LIN {X 0,Y 202.976,Z 342.677,A -85,B 0,C 180,E1 -21997.686,E2 -21997.686} C_VEL
LIN {X 0,Y 206.775,Z 348.376,A -85,B 0,C 180,E1 -21999.696,E2 -21999.696} C_VEL
LIN {X 0,Y 211.34,Z 355.755,A -85,B 0,C 180,E1 -22001.921,E2 -22001.921} C_VEL
LIN {X 0,Y 216.534,Z 364.56,A -85,B 0,C 180,E1 -22004.233,E2 -22004.233} C_VEL
LIN {X 0,Y 221.924,Z 374.855,A -85,B 0,C 180,E1 -22006.449,E2 -22006.449} C_VEL
LIN {X 0,Y 227.529,Z 386.979,A -85,B 0,C 180,E1 -22008.613,E2 -22008.613} C_VEL
LIN {X 0,Y 230.022,Z 393.221,A -85,B 0,C 180,E1 -22009.55,E2 -22009.55} C_VEL
LIN {X 0,Y 230.632,Z 398.833,A -85,B 0,C 180,E1 -22009.954,E2 -22009.954} C_VEL
LIN {X 0,Y 229.742,Z 414.651,A -85,B 0,C 180,E1 -22010.427,E2 -22010.427} C_VEL
LIN {X 0,Y 228.926,Z 420.5,A -85,B 0,C 180,E1 -22010.473,E2 -22010.473} C_VEL
LIN {X 0,Y 223.579,Z 439.513,A -85,B 0,C 180,E1 -22010.007,E2 -22010.007} C_VEL
LIN {X 0,Y 222.491,Z 445.308,A -85,B 0,C 180,E1 -22010.121,E2 -22010.121} C_VEL
LIN {X 0,Y 220.529,Z 457.934,A -85,B 0,C 180,E1 -22010.845,E2 -22010.845} C_VEL
LIN {X 0,Y 217.724,Z 470.431,A -85,B 0,C 180,E1 -22011.877,E2 -22011.877} C_VEL
LIN {X 0,Y 214.297,Z 482.437,A -85,B 0,C 180,E1 -22013.235,E2 -22013.235} C_VEL
LIN {X 0,Y 210.551,Z 493.18,A -85,B 0,C 180,E1 -22014.844,E2 -22014.844} C_VEL
LIN {X 0,Y 206.238,Z 503.921,A -85,B 0,C 180,E1 -22016.958,E2 -22016.958} C_VEL
LIN {X 0,Y 202.158,Z 512.677,A -85,B 0,C 180,E1 -22019.149,E2 -22019.149} C_VEL
LIN {X 0,Y 197.802,Z 521.235,A -85,B 0,C 180,E1 -22021.914,E2 -22021.914} C_VEL
LIN {X 0,Y 193.915,Z 528.409,A -85,B 0,C 180,E1 -22024.968,E2 -22024.968} C_VEL
LIN {X 0,Y 190.389,Z 534.447,A -85,B 0,C 180,E1 -22028.336,E2 -22028.336} C_VEL
LIN {X 0,Y 187.771,Z 538.634,A -85,B 0,C 180,E1 -22031.448,E2 -22031.448} C_VEL
LIN {X 0,Y 185.687,Z 541.79,A -85,B 0,C 180,E1 -22034.635,E2 -22034.635} C_VEL
LIN {X 0,Y 184.75,Z 543.382,A -85,B 0,C 180,E1 -22036.805,E2 -22036.805} C_VEL
LIN {X 0,Y 184.038,Z 544.562,A -85,B 0,C 180,E1 -22038.991,E2 -22038.991} C_VEL
LIN {X 0,Y 183.222,Z 545.704,A -85,B 0,C 180,E1 -22043.391,E2 -22043.391} C_VEL
LIN {X 0,Y 183.133,Z 545.653,A -85,B 0,C 180,E1 -22046.191,E2 -22046.191} C_VEL
LIN {X 0,Y 183.342,Z 544.51,A -85,B 0,C 180,E1 -22049.998,E2 -22049.998} C_VEL
LIN {X 0,Y 183.16,Z 541.988,A -85,B 0,C 180,E1 -22053.935,E2 -22053.935} C_VEL
LIN {X 0,Y 183.374,Z 538.253,A -85,B 0,C 180,E1 -22057.707,E2 -22057.707} C_VEL
LIN {X 0,Y 183.903,Z 533.789,A -85,B 0,C 180,E1 -22061.014,E2 -22061.014} C_VEL
LIN {X 0,Y 184.844,Z 528.091,A -85,B 0,C 180,E1 -22064.306,E2 -22064.306} C_VEL
LIN {X 0,Y 186.496,Z 520.949,A -85,B 0,C 180,E1 -22067.544,E2 -22067.544} C_VEL
LIN {X 0,Y 188.388,Z 512.541,A -85,B 0,C 180,E1 -22070.564,E2 -22070.564} C_VEL
LIN {X 0,Y 189.713,Z 506.711,A -85,B 0,C 180,E1 -22072.314,E2 -22072.314} C_VEL
LIN {X 0,Y 191.746,Z 497.383,A -85,B 0,C 180,E1 -22074.638,E2 -22074.638} C_VEL
LIN {X 0,Y 193.876,Z 487.221,A -85,B 0,C 180,E1 -22076.651,E2 -22076.651} C_VEL
LIN {X 0,Y 196.128,Z 476.194,A -85,B 0,C 180,E1 -22078.344,E2 -22078.344} C_VEL
LIN {X 0,Y 197.847,Z 465.063,A -85,B 0,C 180,E1 -22079.674,E2 -22079.674} C_VEL
LIN {X 0,Y 199.457,Z 452.039,A -85,B 0,C 180,E1 -22080.796,E2 -22080.796} C_VEL
LIN {X 0,Y 200.468,Z 439.102,A -85,B 0,C 180,E1 -22081.503,E2 -22081.503} C_VEL
LIN {X 0,Y 202.387,Z 390.412,A -85,B 0,C 180,E1 -22083.182,E2 -22083.182} C_VEL
LIN {X 0,Y 199.567,Z 364.019,A -85,B 0,C 180,E1 -22084.672,E2 -22084.672} C_VEL
LIN {X 0,Y 193.84,Z 348.784,A -85,B 0,C 180,E1 -22086.254,E2 -22086.254} C_VEL
LIN {X 0,Y 188.083,Z 335.728,A -85,B 0,C 180,E1 -22087.863,E2 -22087.863} C_VEL
LIN {X 0,Y 186.801,Z 332.704,A -85,B 0,C 180,E1 -22088.273,E2 -22088.273} C_VEL
LIN {X 0,Y 185.491,Z 327.376,A -85,B 0,C 180,E1 -22091.228,E2 -22091.228} C_VEL
LIN {X 0,Y 185.456,Z 327.385,A -85,B 0,C 180,E1 -22096.053,E2 -22096.053} C_VEL
LIN {X 0,Y 185.484,Z 327.371,A -85,B 0,C 180,E1 -22099.9,E2 -22099.9} C_VEL
LIN {X 0,Y 185.539,Z 327.374,A -85,B 0,C 180,E1 -22102.695,E2 -22102.695} C_VEL
LIN {X 0,Y 185.54,Z 327.368,A -85,B 0,C 180,E1 -22107.974,E2 -22107.974} C_VEL
LIN {X 0,Y 185.577,Z 327.366,A -85,B 0,C 180,E1 -22110.575,E2 -22110.575} C_VEL
LIN {X 0,Y 185.582,Z 327.364,A -85,B 0,C 180,E1 -22115.382,E2 -22115.382} C_VEL
LIN {X 0,Y 185.601,Z 327.359,A -85,B 0,C 180,E1 -22120.075,E2 -22120.075} C_VEL
LIN {X 0,Y 185.693,Z 327.34,A -85,B 0,C 180,E1 -22124.637,E2 -22124.637} C_VEL
LIN {X 0,Y 185.918,Z 327.324,A -85,B 0,C 180,E1 -22129.359,E2 -22129.359} C_VEL
LIN {X 0,Y 185.954,Z 327.292,A -85,B 0,C 180,E1 -22133.49,E2 -22133.49} C_VEL
LIN {X 0,Y 186.201,Z 327.285,A -85,B 0,C 180,E1 -22137.837,E2 -22137.837} C_VEL
LIN {X 0,Y 186.399,Z 327.265,A -85,B 0,C 180,E1 -22140,E2 -22140} C_VEL
LIN {X 0,Y 185.905,Z 327.305,A -85,B 0,C 180,E1 -22144.336,E2 -22144.336} C_VEL
LIN {X 0,Y 185.97,Z 327.304,A -85,B 0,C 180,E1 -22148.695,E2 -22148.695} C_VEL
LIN {X 0,Y 185.723,Z 327.348,A -85,B 0,C 180,E1 -22153.124,E2 -22153.124} C_VEL
LIN {X 0,Y 185.684,Z 327.353,A -85,B 0,C 180,E1 -22157.626,E2 -22157.626} C_VEL
LIN {X 0,Y 185.575,Z 327.362,A -85,B 0,C 180,E1 -22162.254,E2 -22162.254} C_VEL
LIN {X 0,Y 185.555,Z 327.364,A -85,B 0,C 180,E1 -22167.033,E2 -22167.033} C_VEL
LIN {X 0,Y 185.574,Z 327.364,A -85,B 0,C 180,E1 -22169.494,E2 -22169.494} C_VEL
LIN {X 0,Y 185.494,Z 327.372,A -85,B 0,C 180,E1 -22174.634,E2 -22174.634} C_VEL
LIN {X 0,Y 185.495,Z 327.375,A -85,B 0,C 180,E1 -22177.316,E2 -22177.316} C_VEL
LIN {X 0,Y 185.456,Z 327.38,A -85,B 0,C 180,E1 -22180.723,E2 -22180.723} C_VEL
LIN {X 0,Y 185.451,Z 327.382,A -85,B 0,C 180,E1 -22186.058,E2 -22186.058} C_VEL
LIN {X 0,Y 185.452,Z 327.382,A -85,B 0,C 180,E1 -22189.894,E2 -22189.894} C_VEL
LIN {X 0,Y 185.497,Z 327.375,A -85,B 0,C 180,E1 -22192.716,E2 -22192.716} C_VEL
LIN {X 0,Y 185.528,Z 327.375,A -85,B 0,C 180,E1 -22197.974,E2 -22197.974} C_VEL
LIN {X 0,Y 185.545,Z 327.368,A -85,B 0,C 180,E1 -22200.597,E2 -22200.597} C_VEL
LIN {X 0,Y 185.622,Z 327.361,A -85,B 0,C 180,E1 -22205.853,E2 -22205.853} C_VEL
LIN {X 0,Y 186.53,Z 330.059,A -85,B 0,C 180,E1 -22206.184,E2 -22206.184} C_VEL
LIN {X 0,Y 189.459,Z 335.059,A -85,B 0,C 180,E1 -22206.964,E2 -22206.964} C_VEL
LIN {X 0,Y 198.448,Z 352.648,A -85,B 0,C 180,E1 -22209.284,E2 -22209.284} C_VEL
LIN {X 0,Y 202.191,Z 362.446,A -85,B 0,C 180,E1 -22210.275,E2 -22210.275} C_VEL
LIN {X 0,Y 203.501,Z 366.519,A -85,B 0,C 180,E1 -22210.637,E2 -22210.637} C_VEL
LIN {X 0,Y 200.596,Z 428.694,A -85,B 0,C 180,E1 -22212.741,E2 -22212.741} C_VEL
LIN {X 0,Y 199.469,Z 442.513,A -85,B 0,C 180,E1 -22213.63,E2 -22213.63} C_VEL
LIN {X 0,Y 197.838,Z 454.998,A -85,B 0,C 180,E1 -22214.814,E2 -22214.814} C_VEL
LIN {X 0,Y 196.174,Z 466.075,A -85,B 0,C 180,E1 -22216.272,E2 -22216.272} C_VEL
LIN {X 0,Y 194.083,Z 478.007,A -85,B 0,C 180,E1 -22218.331,E2 -22218.331} C_VEL
LIN {X 0,Y 191.896,Z 488.043,A -85,B 0,C 180,E1 -22220.516,E2 -22220.516} C_VEL
LIN {X 0,Y 189.694,Z 497.422,A -85,B 0,C 180,E1 -22223.086,E2 -22223.086} C_VEL
LIN {X 0,Y 187.523,Z 506.483,A -85,B 0,C 180,E1 -22226.241,E2 -22226.241} C_VEL
LIN {X 0,Y 185.812,Z 513.787,A -85,B 0,C 180,E1 -22229.46,E2 -22229.46} C_VEL
LIN {X 0,Y 184.73,Z 518.72,A -85,B 0,C 180,E1 -22232.182,E2 -22232.182} C_VEL
LIN {X 0,Y 183.835,Z 523.649,A -85,B 0,C 180,E1 -22235.588,E2 -22235.588} C_VEL
LIN {X 0,Y 183.199,Z 527.201,A -85,B 0,C 180,E1 -22238.828,E2 -22238.828} C_VEL
LIN {X 0,Y 182.945,Z 529.103,A -85,B 0,C 180,E1 -22241.076,E2 -22241.076} C_VEL
LIN {X 0,Y 182.886,Z 530.525,A -85,B 0,C 180,E1 -22243.332,E2 -22243.332} C_VEL
LIN {X 0,Y 183.019,Z 531.784,A -85,B 0,C 180,E1 -22246.257,E2 -22246.257} C_VEL
LIN {X 0,Y 183.544,Z 532.345,A -85,B 0,C 180,E1 -22250.16,E2 -22250.16} C_VEL
LIN {X 0,Y 184.788,Z 531.648,A -85,B 0,C 180,E1 -22254.106,E2 -22254.106} C_VEL
LIN {X 0,Y 186.017,Z 530.363,A -85,B 0,C 180,E1 -22256.962,E2 -22256.962} C_VEL
LIN {X 0,Y 188.528,Z 527.22,A -85,B 0,C 180,E1 -22260.973,E2 -22260.973} C_VEL
LIN {X 0,Y 191.528,Z 522.851,A -85,B 0,C 180,E1 -22264.665,E2 -22264.665} C_VEL
LIN {X 0,Y 194.823,Z 517.679,A -85,B 0,C 180,E1 -22267.826,E2 -22267.826} C_VEL
LIN {X 0,Y 198.597,Z 511.056,A -85,B 0,C 180,E1 -22270.897,E2 -22270.897} C_VEL
LIN {X 0,Y 202.949,Z 502.708,A -85,B 0,C 180,E1 -22273.837,E2 -22273.837} C_VEL
LIN {X 0,Y 206.95,Z 494.106,A -85,B 0,C 180,E1 -22276.192,E2 -22276.192} C_VEL
LIN {X 0,Y 211.188,Z 483.825,A -85,B 0,C 180,E1 -22278.361,E2 -22278.361} C_VEL
LIN {X 0,Y 214.941,Z 472.663,A -85,B 0,C 180,E1 -22280.21,E2 -22280.21} C_VEL
LIN {X 0,Y 218.243,Z 460.818,A -85,B 0,C 180,E1 -22281.705,E2 -22281.705} C_VEL
LIN {X 0,Y 220.989,Z 448.028,A -85,B 0,C 180,E1 -22282.878,E2 -22282.878} C_VEL
LIN {X 0,Y 222.908,Z 435.07,A -85,B 0,C 180,E1 -22283.724,E2 -22283.724} C_VEL
LIN {X 0,Y 224.059,Z 422.51,A -85,B 0,C 180,E1 -22284.221,E2 -22284.221} C_VEL
LIN {X 0,Y 226.252,Z 387.885,A -85,B 0,C 180,E1 -22285.23,E2 -22285.23} C_VEL
LIN {X 0,Y 221.111,Z 377.012,A -85,B 0,C 180,E1 -22287.225,E2 -22287.225} C_VEL
LIN {X 0,Y 216.185,Z 368.359,A -85,B 0,C 180,E1 -22289.222,E2 -22289.222} C_VEL
LIN {X 0,Y 208.7,Z 357.089,A -85,B 0,C 180,E1 -22292.547,E2 -22292.547} C_VEL
LIN {X 0,Y 205.082,Z 352.229,A -85,B 0,C 180,E1 -22294.313,E2 -22294.313} C_VEL
LIN {X 0,Y 202.026,Z 348.124,A -85,B 0,C 180,E1 -22295.924,E2 -22295.924} C_VEL
LIN {X 0,Y 199.302,Z 344.502,A -85,B 0,C 180,E1 -22297.467,E2 -22297.467} C_VEL
LIN {X 0,Y 198.265,Z 343.307,A -85,B 0,C 180,E1 -22298.072,E2 -22298.072} C_VEL
LIN {X 0,Y 195.827,Z 340.436,A -85,B 0,C 180,E1 -22299.586,E2 -22299.586} C_VEL
LIN {X 0,Y 194.758,Z 338.66,A -85,B 0,C 180,E1 -22300.329,E2 -22300.329} C_VEL
LIN {X 0,Y 192.265,Z 336.46,A -85,B 0,C 180,E1 -22302.006,E2 -22302.006} C_VEL
LIN {X 0,Y 190.4,Z 333.17,A -85,B 0,C 180,E1 -22303.515,E2 -22303.515} C_VEL
LIN {X 0,Y 187.845,Z 331.569,A -85,B 0,C 180,E1 -22305.51,E2 -22305.51} C_VEL
LIN {X 0,Y 186.355,Z 329.381,A -85,B 0,C 180,E1 -22306.922,E2 -22306.922} C_VEL
LIN {X 0,Y 185.829,Z 327.334,A -85,B 0,C 180,E1 -22307.648,E2 -22307.648} C_VEL
LIN {X 0,Y 186.017,Z 327.297,A -85,B 0,C 180,E1 -22311.308,E2 -22311.308} C_VEL
LIN {X 0,Y 186.209,Z 327.286,A -85,B 0,C 180,E1 -22317.837,E2 -22317.837} C_VEL
LIN {X 0,Y 186.407,Z 327.247,A -85,B 0,C 180,E1 -22320,E2 -22320} C_VEL
LIN {X 0,Y 185.928,Z 327.314,A -85,B 0,C 180,E1 -22324.336,E2 -22324.336} C_VEL
LIN {X 0,Y 186.032,Z 327.309,A -85,B 0,C 180,E1 -22328.691,E2 -22328.691} C_VEL
LIN {X 0,Y 185.742,Z 327.338,A -85,B 0,C 180,E1 -22333.122,E2 -22333.122} C_VEL
LIN {X 0,Y 185.693,Z 327.342,A -85,B 0,C 180,E1 -22337.625,E2 -22337.625} C_VEL
LIN {X 0,Y 185.636,Z 327.442,A -85,B 0,C 180,E1 -22344.015,E2 -22344.015} C_VEL
LIN {X 0,Y 186.178,Z 329.465,A -85,B 0,C 180,E1 -22346.481,E2 -22346.481} C_VEL
LIN {X 0,Y 190.887,Z 335.576,A -85,B 0,C 180,E1 -22350.567,E2 -22350.567} C_VEL
LIN {X 0,Y 191.989,Z 336.995,A -85,B 0,C 180,E1 -22351.403,E2 -22351.403} C_VEL
LIN {X 0,Y 196.832,Z 343.634,A -85,B 0,C 180,E1 -22354.743,E2 -22354.743} C_VEL
LIN {X 0,Y 201.039,Z 349.855,A -85,B 0,C 180,E1 -22357.275,E2 -22357.275} C_VEL
LIN {X 0,Y 204.668,Z 355.514,A -85,B 0,C 180,E1 -22359.259,E2 -22359.259} C_VEL
LIN {X 0,Y 208.635,Z 362.026,A -85,B 0,C 180,E1 -22361.26,E2 -22361.26} C_VEL
LIN {X 0,Y 213.158,Z 370,A -85,B 0,C 180,E1 -22363.374,E2 -22363.374} C_VEL
LIN {X 0,Y 217.819,Z 379.047,A -85,B 0,C 180,E1 -22365.401,E2 -22365.401} C_VEL
LIN {X 0,Y 223.263,Z 391.128,A -85,B 0,C 180,E1 -22367.626,E2 -22367.626} C_VEL
LIN {X 0,Y 225.342,Z 396.563,A -85,B 0,C 180,E1 -22368.462,E2 -22368.462} C_VEL
LIN {X 0,Y 225.627,Z 400.453,A -85,B 0,C 180,E1 -22368.72,E2 -22368.72} C_VEL
LIN {X 0,Y 222.891,Z 441.6,A -85,B 0,C 180,E1 -22369.961,E2 -22369.961} C_VEL
LIN {X 0,Y 222.491,Z 445.308,A -85,B 0,C 180,E1 -22370.121,E2 -22370.121} C_VEL
LIN {X 0,Y 221.225,Z 451.068,A -85,B 0,C 180,E1 -22370.272,E2 -22370.272} C_VEL
LIN {X 0,Y 217.492,Z 460.287,A -85,B 0,C 180,E1 -22370.327,E2 -22370.327} C_VEL
LIN {X 0,Y 213.343,Z 469.24,A -85,B 0,C 180,E1 -22370.562,E2 -22370.562} C_VEL
LIN {X 0,Y 211.432,Z 474.575,A -85,B 0,C 180,E1 -22371.002,E2 -22371.002} C_VEL
LIN {X 0,Y 207.686,Z 486.208,A -85,B 0,C 180,E1 -22372.474,E2 -22372.474} C_VEL
LIN {X 0,Y 203.429,Z 497.309,A -85,B 0,C 180,E1 -22374.338,E2 -22374.338} C_VEL
LIN {X 0,Y 199.469,Z 506.297,A -85,B 0,C 180,E1 -22376.293,E2 -22376.293} C_VEL
LIN {X 0,Y 195.342,Z 514.566,A -85,B 0,C 180,E1 -22378.554,E2 -22378.554} C_VEL
LIN {X 0,Y 190.845,Z 522.685,A -85,B 0,C 180,E1 -22381.396,E2 -22381.396} C_VEL
LIN {X 0,Y 187.272,Z 528.934,A -85,B 0,C 180,E1 -22384.248,E2 -22384.248} C_VEL
LIN {X 0,Y 183.801,Z 534.5,A -85,B 0,C 180,E1 -22387.518,E2 -22387.518} C_VEL
LIN {X 0,Y 181.045,Z 538.613,A -85,B 0,C 180,E1 -22390.732,E2 -22390.732} C_VEL
LIN {X 0,Y 178.819,Z 541.7,A -85,B 0,C 180,E1 -22394.03,E2 -22394.03} C_VEL
LIN {X 0,Y 177.81,Z 543.256,A -85,B 0,C 180,E1 -22396.28,E2 -22396.28} C_VEL
LIN {X 0,Y 176.474,Z 545.102,A -85,B 0,C 180,E1 -22400.832,E2 -22400.832} C_VEL
LIN {X 0,Y 176.067,Z 545.429,A -85,B 0,C 180,E1 -22405.419,E2 -22405.419} C_VEL
LIN {X 0,Y 176.083,Z 544.99,A -85,B 0,C 180,E1 -22407.711,E2 -22407.711} C_VEL
LIN {X 0,Y 176.26,Z 544.136,A -85,B 0,C 180,E1 -22409.998,E2 -22409.998} C_VEL
LIN {X 0,Y 176.072,Z 541.836,A -85,B 0,C 180,E1 -22413.726,E2 -22413.726} C_VEL
LIN {X 0,Y 176.329,Z 537.744,A -85,B 0,C 180,E1 -22418.017,E2 -22418.017} C_VEL
LIN {X 0,Y 176.903,Z 533.205,A -85,B 0,C 180,E1 -22421.456,E2 -22421.456} C_VEL
LIN {X 0,Y 178.177,Z 526.286,A -85,B 0,C 180,E1 -22425.439,E2 -22425.439} C_VEL
LIN {X 0,Y 179.936,Z 518.76,A -85,B 0,C 180,E1 -22428.796,E2 -22428.796} C_VEL
LIN {X 0,Y 181.55,Z 512.072,A -85,B 0,C 180,E1 -22431.213,E2 -22431.213} C_VEL
LIN {X 0,Y 183.619,Z 503.724,A -85,B 0,C 180,E1 -22433.694,E2 -22433.694} C_VEL
LIN {X 0,Y 185.818,Z 493.804,A -85,B 0,C 180,E1 -22436.081,E2 -22436.081} C_VEL
LIN {X 0,Y 188.191,Z 482.899,A -85,B 0,C 180,E1 -22438.128,E2 -22438.128} C_VEL
LIN {X 0,Y 190.287,Z 471.631,A -85,B 0,C 180,E1 -22439.753,E2 -22439.753} C_VEL
LIN {X 0,Y 192.142,Z 459.067,A -85,B 0,C 180,E1 -22441.106,E2 -22441.106} C_VEL
LIN {X 0,Y 193.655,Z 446.042,A -85,B 0,C 180,E1 -22442.055,E2 -22442.055} C_VEL
LIN {X 0,Y 194.592,Z 430.245,A -85,B 0,C 180,E1 -22442.724,E2 -22442.724} C_VEL
LIN {X 0,Y 196.074,Z 391.001,A -85,B 0,C 180,E1 -22444.113,E2 -22444.113} C_VEL
LIN {X 0,Y 193.564,Z 366.443,A -85,B 0,C 180,E1 -22445.55,E2 -22445.55} C_VEL
LIN {X 0,Y 187.863,Z 351.135,A -85,B 0,C 180,E1 -22447.221,E2 -22447.221} C_VEL
LIN {X 0,Y 182.501,Z 338.983,A -85,B 0,C 180,E1 -22448.806,E2 -22448.806} C_VEL
LIN {X 0,Y 179.48,Z 332.395,A -85,B 0,C 180,E1 -22449.769,E2 -22449.769} C_VEL
LIN {X 0,Y 178.416,Z 328.259,A -85,B 0,C 180,E1 -22452.227,E2 -22452.227} C_VEL
LIN {X 0,Y 178.39,Z 328.264,A -85,B 0,C 180,E1 -22455.162,E2 -22455.162} C_VEL
LIN {X 0,Y 178.406,Z 328.26,A -85,B 0,C 180,E1 -22458.455,E2 -22458.455} C_VEL
LIN {X 0,Y 178.459,Z 328.252,A -85,B 0,C 180,E1 -22461.961,E2 -22461.961} C_VEL
LIN {X 0,Y 178.486,Z 328.251,A -85,B 0,C 180,E1 -22466.547,E2 -22466.547} C_VEL
LIN {X 0,Y 178.517,Z 328.246,A -85,B 0,C 180,E1 -22470.005,E2 -22470.005} C_VEL
LIN {X 0,Y 178.529,Z 328.243,A -85,B 0,C 180,E1 -22474.875,E2 -22474.875} C_VEL
LIN {X 0,Y 178.617,Z 328.221,A -85,B 0,C 180,E1 -22480.783,E2 -22480.783} C_VEL
LIN {X 0,Y 178.674,Z 328.224,A -85,B 0,C 180,E1 -22486.349,E2 -22486.349} C_VEL
LIN {X 0,Y 178.953,Z 328.182,A -85,B 0,C 180,E1 -22490.962,E2 -22490.962} C_VEL
LIN {X 0,Y 179.146,Z 328.162,A -85,B 0,C 180,E1 -22497.752,E2 -22497.752} C_VEL
LIN {X 0,Y 179.363,Z 328.141,A -85,B 0,C 180,E1 -22500,E2 -22500} C_VEL
LIN {X 0,Y 178.852,Z 328.18,A -85,B 0,C 180,E1 -22504.508,E2 -22504.508} C_VEL
LIN {X 0,Y 178.9,Z 328.188,A -85,B 0,C 180,E1 -22509.041,E2 -22509.041} C_VEL
LIN {X 0,Y 178.651,Z 328.23,A -85,B 0,C 180,E1 -22513.653,E2 -22513.653} C_VEL
LIN {X 0,Y 178.616,Z 328.235,A -85,B 0,C 180,E1 -22519.216,E2 -22519.216} C_VEL
LIN {X 0,Y 178.514,Z 328.247,A -85,B 0,C 180,E1 -22525.115,E2 -22525.115} C_VEL
LIN {X 0,Y 178.496,Z 328.249,A -85,B 0,C 180,E1 -22530.788,E2 -22530.788} C_VEL
LIN {X 0,Y 178.48,Z 328.243,A -85,B 0,C 180,E1 -22534.221,E2 -22534.221} C_VEL
LIN {X 0,Y 178.382,Z 328.256,A -85,B 0,C 180,E1 -22539.078,E2 -22539.078} C_VEL
LIN {X 0,Y 178.388,Z 328.262,A -85,B 0,C 180,E1 -22542.048,E2 -22542.048} C_VEL
LIN {X 0,Y 178.387,Z 328.26,A -85,B 0,C 180,E1 -22545.167,E2 -22545.167} C_VEL
LIN {X 0,Y 178.393,Z 328.258,A -85,B 0,C 180,E1 -22548.463,E2 -22548.463} C_VEL
LIN {X 0,Y 178.416,Z 328.258,A -85,B 0,C 180,E1 -22553.784,E2 -22553.784} C_VEL
LIN {X 0,Y 178.481,Z 328.25,A -85,B 0,C 180,E1 -22556.548,E2 -22556.548} C_VEL
LIN {X 0,Y 178.442,Z 328.258,A -85,B 0,C 180,E1 -22561.798,E2 -22561.798} C_VEL
LIN {X 0,Y 178.471,Z 328.254,A -85,B 0,C 180,E1 -22564.396,E2 -22564.396} C_VEL
LIN {X 0,Y 179.635,Z 331.322,A -85,B 0,C 180,E1 -22564.841,E2 -22564.841} C_VEL
LIN {X 0,Y 181.116,Z 333.578,A -85,B 0,C 180,E1 -22565.259,E2 -22565.259} C_VEL
LIN {X 0,Y 188.684,Z 347.58,A -85,B 0,C 180,E1 -22567.374,E2 -22567.374} C_VEL
LIN {X 0,Y 194.402,Z 359.697,A -85,B 0,C 180,E1 -22568.908,E2 -22568.908} C_VEL
LIN {X 0,Y 197.197,Z 367.778,A -85,B 0,C 180,E1 -22569.707,E2 -22569.707} C_VEL
LIN {X 0,Y 194.265,Z 428.652,A -85,B 0,C 180,E1 -22571.819,E2 -22571.819} C_VEL
LIN {X 0,Y 193.106,Z 442.237,A -85,B 0,C 180,E1 -22572.702,E2 -22572.702} C_VEL
LIN {X 0,Y 191.463,Z 454.568,A -85,B 0,C 180,E1 -22573.885,E2 -22573.885} C_VEL
LIN {X 0,Y 189.576,Z 466.631,A -85,B 0,C 180,E1 -22575.51,E2 -22575.51} C_VEL
LIN {X 0,Y 187.362,Z 478.715,A -85,B 0,C 180,E1 -22577.676,E2 -22577.676} C_VEL
LIN {X 0,Y 184.899,Z 489.517,A -85,B 0,C 180,E1 -22580.153,E2 -22580.153} C_VEL
LIN {X 0,Y 182.61,Z 498.657,A -85,B 0,C 180,E1 -22582.816,E2 -22582.816} C_VEL
LIN {X 0,Y 180.395,Z 507.556,A -85,B 0,C 180,E1 -22586.092,E2 -22586.092} C_VEL
LIN {X 0,Y 178.661,Z 514.692,A -85,B 0,C 180,E1 -22589.438,E2 -22589.438} C_VEL
LIN {X 0,Y 177.261,Z 521.194,A -85,B 0,C 180,E1 -22593.411,E2 -22593.411} C_VEL
LIN {X 0,Y 176.451,Z 525.496,A -85,B 0,C 180,E1 -22596.864,E2 -22596.864} C_VEL
LIN {X 0,Y 176.036,Z 527.793,A -85,B 0,C 180,E1 -22599.191,E2 -22599.191} C_VEL
LIN {X 0,Y 175.812,Z 529.596,A -85,B 0,C 180,E1 -22601.531,E2 -22601.531} C_VEL
LIN {X 0,Y 175.817,Z 530.965,A -85,B 0,C 180,E1 -22603.879,E2 -22603.879} C_VEL
LIN {X 0,Y 175.932,Z 532.034,A -85,B 0,C 180,E1 -22606.516,E2 -22606.516} C_VEL
LIN {X 0,Y 176.622,Z 532.594,A -85,B 0,C 180,E1 -22610.986,E2 -22610.986} C_VEL
LIN {X 0,Y 177.852,Z 531.944,A -85,B 0,C 180,E1 -22614.65,E2 -22614.65} C_VEL
LIN {X 0,Y 179.419,Z 530.414,A -85,B 0,C 180,E1 -22618.039,E2 -22618.039} C_VEL
LIN {X 0,Y 181.842,Z 527.571,A -85,B 0,C 180,E1 -22621.757,E2 -22621.757} C_VEL
LIN {X 0,Y 184.399,Z 524.145,A -85,B 0,C 180,E1 -22624.87,E2 -22624.87} C_VEL
LIN {X 0,Y 187.794,Z 519.172,A -85,B 0,C 180,E1 -22628.195,E2 -22628.195} C_VEL
LIN {X 0,Y 191.616,Z 513.002,A -85,B 0,C 180,E1 -22631.316,E2 -22631.316} C_VEL
LIN {X 0,Y 195.502,Z 506.083,A -85,B 0,C 180,E1 -22634.03,E2 -22634.03} C_VEL
LIN {X 0,Y 199.294,Z 498.739,A -85,B 0,C 180,E1 -22636.297,E2 -22636.297} C_VEL
LIN {X 0,Y 203.725,Z 489.175,A -85,B 0,C 180,E1 -22638.62,E2 -22638.62} C_VEL
LIN {X 0,Y 207.871,Z 478.431,A -85,B 0,C 180,E1 -22640.646,E2 -22640.646} C_VEL
LIN {X 0,Y 211.251,Z 467.915,A -85,B 0,C 180,E1 -22642.198,E2 -22642.198} C_VEL
LIN {X 0,Y 214.396,Z 456.043,A -85,B 0,C 180,E1 -22643.529,E2 -22643.529} C_VEL
LIN {X 0,Y 216.977,Z 442.644,A -85,B 0,C 180,E1 -22644.609,E2 -22644.609} C_VEL
LIN {X 0,Y 218.542,Z 430.622,A -85,B 0,C 180,E1 -22645.266,E2 -22645.266} C_VEL
LIN {X 0,Y 221.279,Z 392.274,A -85,B 0,C 180,E1 -22646.427,E2 -22646.427} C_VEL
LIN {X 0,Y 221.249,Z 390.383,A -85,B 0,C 180,E1 -22646.528,E2 -22646.528} C_VEL
LIN {X 0,Y 216.708,Z 380.728,A -85,B 0,C 180,E1 -22648.402,E2 -22648.402} C_VEL
LIN {X 0,Y 212.653,Z 373.521,A -85,B 0,C 180,E1 -22650.15,E2 -22650.15} C_VEL
LIN {X 0,Y 205.829,Z 362.903,A -85,B 0,C 180,E1 -22653.341,E2 -22653.341} C_VEL
LIN {X 0,Y 201.746,Z 357.346,A -85,B 0,C 180,E1 -22655.44,E2 -22655.44} C_VEL
LIN {X 0,Y 199.298,Z 354.01,A -85,B 0,C 180,E1 -22656.803,E2 -22656.803} C_VEL
LIN {X 0,Y 196.075,Z 349.69,A -85,B 0,C 180,E1 -22658.74,E2 -22658.74} C_VEL
LIN {X 0,Y 193.404,Z 346.364,A -85,B 0,C 180,E1 -22660.488,E2 -22660.488} C_VEL
LIN {X 0,Y 192.637,Z 345.118,A -85,B 0,C 180,E1 -22661.043,E2 -22661.043} C_VEL
LIN {X 0,Y 189.931,Z 342.39,A -85,B 0,C 180,E1 -22662.989,E2 -22662.989} C_VEL
LIN {X 0,Y 188.374,Z 339.794,A -85,B 0,C 180,E1 -22664.306,E2 -22664.306} C_VEL
LIN {X 0,Y 185.67,Z 337.577,A -85,B 0,C 180,E1 -22666.594,E2 -22666.594} C_VEL
LIN {X 0,Y 184.246,Z 334.996,A -85,B 0,C 180,E1 -22668.099,E2 -22668.099} C_VEL
LIN {X 0,Y 183.989,Z 334.194,A -85,B 0,C 180,E1 -22668.431,E2 -22668.431} C_VEL
LIN {X 0,Y 180.993,Z 332.351,A -85,B 0,C 180,E1 -22671.768,E2 -22671.768} C_VEL
LIN {X 0,Y 179.279,Z 329.828,A -85,B 0,C 180,E1 -22674.376,E2 -22674.376} C_VEL
LIN {X 0,Y 178.883,Z 328.183,A -85,B 0,C 180,E1 -22675.352,E2 -22675.352} C_VEL
LIN {X 0,Y 179.371,Z 328.123,A -85,B 0,C 180,E1 -22680,E2 -22680} C_VEL
LIN {X 0,Y 178.877,Z 328.19,A -85,B 0,C 180,E1 -22684.507,E2 -22684.507} C_VEL
LIN {X 0,Y 178.981,Z 328.185,A -85,B 0,C 180,E1 -22689.037,E2 -22689.037} C_VEL
LIN {X 0,Y 178.668,Z 328.227,A -85,B 0,C 180,E1 -22693.651,E2 -22693.651} C_VEL
LIN {X 0,Y 178.672,Z 328.381,A -85,B 0,C 180,E1 -22697.971,E2 -22697.971} C_VEL
LIN {X 0,Y 179.428,Z 330.827,A -85,B 0,C 180,E1 -22699.548,E2 -22699.548} C_VEL
LIN {X 0,Y 181.291,Z 333.015,A -85,B 0,C 180,E1 -22702.208,E2 -22702.208} C_VEL
LIN {X 0,Y 182.884,Z 334.202,A -85,B 0,C 180,E1 -22704.05,E2 -22704.05} C_VEL
LIN {X 0,Y 184.657,Z 336.322,A -85,B 0,C 180,E1 -22705.956,E2 -22705.956} C_VEL
LIN {X 0,Y 189.82,Z 343.124,A -85,B 0,C 180,E1 -22710.545,E2 -22710.545} C_VEL
LIN {X 0,Y 194.587,Z 349.954,A -85,B 0,C 180,E1 -22714.009,E2 -22714.009} C_VEL
LIN {X 0,Y 198.454,Z 355.887,A -85,B 0,C 180,E1 -22716.459,E2 -22716.459} C_VEL
LIN {X 0,Y 202.153,Z 361.841,A -85,B 0,C 180,E1 -22718.575,E2 -22718.575} C_VEL
LIN {X 0,Y 205.563,Z 367.576,A -85,B 0,C 180,E1 -22720.377,E2 -22720.377} C_VEL
LIN {X 0,Y 211.444,Z 378.37,A -85,B 0,C 180,E1 -22723.231,E2 -22723.231} C_VEL
LIN {X 0,Y 216.853,Z 390.054,A -85,B 0,C 180,E1 -22725.66,E2 -22725.66} C_VEL
LIN {X 0,Y 220.715,Z 399.675,A -85,B 0,C 180,E1 -22727.305,E2 -22727.305} C_VEL
LIN {X 0,Y 220.363,Z 408.095,A -85,B 0,C 180,E1 -22727.612,E2 -22727.612} C_VEL
LIN {X 0,Y 218.001,Z 441.328,A -85,B 0,C 180,E1 -22728.62,E2 -22728.62} C_VEL
LIN {X 0,Y 216.04,Z 455.174,A -85,B 0,C 180,E1 -22729.349,E2 -22729.349} C_VEL
LIN {X 0,Y 213.31,Z 467.826,A -85,B 0,C 180,E1 -22730.33,E2 -22730.33} C_VEL
LIN {X 0,Y 211.432,Z 474.575,A -85,B 0,C 180,E1 -22731.002,E2 -22731.002} C_VEL
LIN {X 0,Y 209.4,Z 479.882,A -85,B 0,C 180,E1 -22731.509,E2 -22731.509} C_VEL
LIN {X 0,Y 204.444,Z 488.182,A -85,B 0,C 180,E1 -22732.132,E2 -22732.132} C_VEL
LIN {X 0,Y 199.168,Z 496.005,A -85,B 0,C 180,E1 -22732.92,E2 -22732.92} C_VEL
LIN {X 0,Y 196.629,Z 500.547,A -85,B 0,C 180,E1 -22733.698,E2 -22733.698} C_VEL
LIN {X 0,Y 191.894,Z 510.21,A -85,B 0,C 180,E1 -22736.045,E2 -22736.045} C_VEL
LIN {X 0,Y 186.922,Z 519.127,A -85,B 0,C 180,E1 -22738.869,E2 -22738.869} C_VEL
LIN {X 0,Y 182.556,Z 526.33,A -85,B 0,C 180,E1 -22741.861,E2 -22741.861} C_VEL
LIN {X 0,Y 179.511,Z 531.215,A -85,B 0,C 180,E1 -22744.489,E2 -22744.489} C_VEL
LIN {X 0,Y 176.209,Z 535.993,A -85,B 0,C 180,E1 -22747.733,E2 -22747.733} C_VEL
LIN {X 0,Y 173.475,Z 539.685,A -85,B 0,C 180,E1 -22751.087,E2 -22751.087} C_VEL
LIN {X 0,Y 171.975,Z 541.61,A -85,B 0,C 180,E1 -22753.376,E2 -22753.376} C_VEL
LIN {X 0,Y 170.875,Z 543.11,A -85,B 0,C 180,E1 -22755.712,E2 -22755.712} C_VEL
LIN {X 0,Y 169.456,Z 544.884,A -85,B 0,C 180,E1 -22760.449,E2 -22760.449} C_VEL
LIN {X 0,Y 168.997,Z 545.14,A -85,B 0,C 180,E1 -22765.227,E2 -22765.227} C_VEL
LIN {X 0,Y 168.996,Z 544.646,A -85,B 0,C 180,E1 -22767.615,E2 -22767.615} C_VEL
LIN {X 0,Y 169.179,Z 543.761,A -85,B 0,C 180,E1 -22769.998,E2 -22769.998} C_VEL
LIN {X 0,Y 169.001,Z 541.626,A -85,B 0,C 180,E1 -22773.573,E2 -22773.573} C_VEL
LIN {X 0,Y 169.154,Z 538.487,A -85,B 0,C 180,E1 -22777.158,E2 -22777.158} C_VEL
LIN {X 0,Y 169.65,Z 534.254,A -85,B 0,C 180,E1 -22780.742,E2 -22780.742} C_VEL
LIN {X 0,Y 170.798,Z 527.781,A -85,B 0,C 180,E1 -22784.901,E2 -22784.901} C_VEL
LIN {X 0,Y 172.554,Z 520.707,A -85,B 0,C 180,E1 -22788.398,E2 -22788.398} C_VEL
LIN {X 0,Y 174.649,Z 512.096,A -85,B 0,C 180,E1 -22791.74,E2 -22791.74} C_VEL
LIN {X 0,Y 177.1,Z 502.68,A -85,B 0,C 180,E1 -22794.623,E2 -22794.623} C_VEL
LIN {X 0,Y 179.134,Z 493.789,A -85,B 0,C 180,E1 -22796.817,E2 -22796.817} C_VEL
LIN {X 0,Y 181.594,Z 482.964,A -85,B 0,C 180,E1 -22798.93,E2 -22798.93} C_VEL
LIN {X 0,Y 183.923,Z 470.777,A -85,B 0,C 180,E1 -22800.734,E2 -22800.734} C_VEL
LIN {X 0,Y 185.888,Z 458.045,A -85,B 0,C 180,E1 -22802.116,E2 -22802.116} C_VEL
LIN {X 0,Y 187.345,Z 445.585,A -85,B 0,C 180,E1 -22803.031,E2 -22803.031} C_VEL
LIN {X 0,Y 188.311,Z 429.669,A -85,B 0,C 180,E1 -22803.719,E2 -22803.719} C_VEL
LIN {X 0,Y 189.825,Z 391.74,A -85,B 0,C 180,E1 -22805.099,E2 -22805.099} C_VEL
LIN {X 0,Y 187.558,Z 368.589,A -85,B 0,C 180,E1 -22806.505,E2 -22806.505} C_VEL
LIN {X 0,Y 180.929,Z 350.966,A -85,B 0,C 180,E1 -22808.566,E2 -22808.566} C_VEL
LIN {X 0,Y 174.142,Z 336.245,A -85,B 0,C 180,E1 -22810.728,E2 -22810.728} C_VEL
LIN {X 0,Y 172.106,Z 332.091,A -85,B 0,C 180,E1 -22811.427,E2 -22811.427} C_VEL
LIN {X 0,Y 171.401,Z 329.133,A -85,B 0,C 180,E1 -22813.277,E2 -22813.277} C_VEL
LIN {X 0,Y 171.34,Z 329.136,A -85,B 0,C 180,E1 -22818.983,E2 -22818.983} C_VEL
LIN {X 0,Y 171.409,Z 329.131,A -85,B 0,C 180,E1 -22822.047,E2 -22822.047} C_VEL
LIN {X 0,Y 171.406,Z 329.132,A -85,B 0,C 180,E1 -22825.085,E2 -22825.085} C_VEL
LIN {X 0,Y 171.444,Z 329.126,A -85,B 0,C 180,E1 -22830.533,E2 -22830.533} C_VEL
LIN {X 0,Y 171.452,Z 329.124,A -85,B 0,C 180,E1 -22835.801,E2 -22835.801} C_VEL
LIN {X 0,Y 171.573,Z 329.096,A -85,B 0,C 180,E1 -22840.871,E2 -22840.871} C_VEL
LIN {X 0,Y 171.587,Z 329.103,A -85,B 0,C 180,E1 -22845.774,E2 -22845.774} C_VEL
LIN {X 0,Y 171.882,Z 329.066,A -85,B 0,C 180,E1 -22850.587,E2 -22850.587} C_VEL
LIN {X 0,Y 171.814,Z 329.056,A -85,B 0,C 180,E1 -22855.308,E2 -22855.308} C_VEL
LIN {X 0,Y 172.325,Z 329.018,A -85,B 0,C 180,E1 -22860,E2 -22860} C_VEL
LIN {X 0,Y 171.8,Z 329.055,A -85,B 0,C 180,E1 -22864.693,E2 -22864.693} C_VEL
LIN {X 0,Y 171.838,Z 329.068,A -85,B 0,C 180,E1 -22869.416,E2 -22869.416} C_VEL
LIN {X 0,Y 171.569,Z 329.108,A -85,B 0,C 180,E1 -22874.228,E2 -22874.228} C_VEL
LIN {X 0,Y 171.536,Z 329.117,A -85,B 0,C 180,E1 -22879.56,E2 -22879.56} C_VEL
LIN {X 0,Y 171.453,Z 329.126,A -85,B 0,C 180,E1 -22885.61,E2 -22885.61} C_VEL
LIN {X 0,Y 171.453,Z 329.127,A -85,B 0,C 180,E1 -22890.598,E2 -22890.598} C_VEL
LIN {X 0,Y 171.387,Z 329.131,A -85,B 0,C 180,E1 -22895.036,E2 -22895.036} C_VEL
LIN {X 0,Y 171.338,Z 329.134,A -85,B 0,C 180,E1 -22898.803,E2 -22898.803} C_VEL
LIN {X 0,Y 171.314,Z 329.137,A -85,B 0,C 180,E1 -22904.22,E2 -22904.22} C_VEL
LIN {X 0,Y 171.326,Z 329.138,A -85,B 0,C 180,E1 -22908.982,E2 -22908.982} C_VEL
LIN {X 0,Y 171.356,Z 329.138,A -85,B 0,C 180,E1 -22912.036,E2 -22912.036} C_VEL
LIN {X 0,Y 171.395,Z 329.137,A -85,B 0,C 180,E1 -22915.095,E2 -22915.095} C_VEL
LIN {X 0,Y 171.407,Z 329.129,A -85,B 0,C 180,E1 -22920.529,E2 -22920.529} C_VEL
LIN {X 0,Y 171.391,Z 329.134,A -85,B 0,C 180,E1 -22922.861,E2 -22922.861} C_VEL
LIN {X 0,Y 172.359,Z 331.901,A -85,B 0,C 180,E1 -22923.245,E2 -22923.245} C_VEL
LIN {X 0,Y 174.03,Z 334.43,A -85,B 0,C 180,E1 -22923.758,E2 -22923.758} C_VEL
LIN {X 0,Y 179.473,Z 343.927,A -85,B 0,C 180,E1 -22925.406,E2 -22925.406} C_VEL
LIN {X 0,Y 187.342,Z 359.622,A -85,B 0,C 180,E1 -22927.662,E2 -22927.662} C_VEL
LIN {X 0,Y 190.563,Z 368.189,A -85,B 0,C 180,E1 -22928.612,E2 -22928.612} C_VEL
LIN {X 0,Y 190.86,Z 370.005,A -85,B 0,C 180,E1 -22928.742,E2 -22928.742} C_VEL
LIN {X 0,Y 187.898,Z 429.773,A -85,B 0,C 180,E1 -22930.898,E2 -22930.898} C_VEL
LIN {X 0,Y 186.677,Z 443.395,A -85,B 0,C 180,E1 -22931.836,E2 -22931.836} C_VEL
LIN {X 0,Y 184.811,Z 456.279,A -85,B 0,C 180,E1 -22933.146,E2 -22933.146} C_VEL
LIN {X 0,Y 182.738,Z 468.763,A -85,B 0,C 180,E1 -22934.955,E2 -22934.955} C_VEL
LIN {X 0,Y 180.454,Z 480.458,A -85,B 0,C 180,E1 -22937.191,E2 -22937.191} C_VEL
LIN {X 0,Y 177.887,Z 490.942,A -85,B 0,C 180,E1 -22939.761,E2 -22939.761} C_VEL
LIN {X 0,Y 175.525,Z 499.894,A -85,B 0,C 180,E1 -22942.525,E2 -22942.525} C_VEL
LIN {X 0,Y 173.262,Z 508.609,A -85,B 0,C 180,E1 -22945.931,E2 -22945.931} C_VEL
LIN {X 0,Y 171.531,Z 515.556,A -85,B 0,C 180,E1 -22949.415,E2 -22949.415} C_VEL
LIN {X 0,Y 170.12,Z 521.941,A -85,B 0,C 180,E1 -22953.554,E2 -22953.554} C_VEL
LIN {X 0,Y 169.284,Z 526.139,A -85,B 0,C 180,E1 -22957.156,E2 -22957.156} C_VEL
LIN {X 0,Y 168.901,Z 528.351,A -85,B 0,C 180,E1 -22959.583,E2 -22959.583} C_VEL
LIN {X 0,Y 168.691,Z 530.086,A -85,B 0,C 180,E1 -22962.025,E2 -22962.025} C_VEL
LIN {X 0,Y 168.721,Z 531.408,A -85,B 0,C 180,E1 -22964.475,E2 -22964.475} C_VEL
LIN {X 0,Y 168.883,Z 532.326,A -85,B 0,C 180,E1 -22966.938,E2 -22966.938} C_VEL
LIN {X 0,Y 169.18,Z 532.788,A -85,B 0,C 180,E1 -22969.412,E2 -22969.412} C_VEL
LIN {X 0,Y 169.74,Z 532.843,A -85,B 0,C 180,E1 -22971.88,E2 -22971.88} C_VEL
LIN {X 0,Y 170.965,Z 532.233,A -85,B 0,C 180,E1 -22975.26,E2 -22975.26} C_VEL
LIN {X 0,Y 172.888,Z 530.464,A -85,B 0,C 180,E1 -22979.198,E2 -22979.198} C_VEL
LIN {X 0,Y 175.203,Z 527.918,A -85,B 0,C 180,E1 -22982.607,E2 -22982.607} C_VEL
LIN {X 0,Y 178.338,Z 523.983,A -85,B 0,C 180,E1 -22986.238,E2 -22986.238} C_VEL
LIN {X 0,Y 182.25,Z 518.562,A -85,B 0,C 180,E1 -22989.838,E2 -22989.838} C_VEL
LIN {X 0,Y 186.083,Z 512.598,A -85,B 0,C 180,E1 -22992.831,E2 -22992.831} C_VEL
LIN {X 0,Y 189.755,Z 506.384,A -85,B 0,C 180,E1 -22995.274,E2 -22995.274} C_VEL
LIN {X 0,Y 194.229,Z 498.013,A -85,B 0,C 180,E1 -22997.884,E2 -22997.884} C_VEL
LIN {X 0,Y 198.907,Z 488.153,A -85,B 0,C 180,E1 -23000.22,E2 -23000.22} C_VEL
LIN {X 0,Y 203.234,Z 477.226,A -85,B 0,C 180,E1 -23002.243,E2 -23002.243} C_VEL
LIN {X 0,Y 206.797,Z 466.238,A -85,B 0,C 180,E1 -23003.819,E2 -23003.819} C_VEL
LIN {X 0,Y 209.692,Z 455.261,A -85,B 0,C 180,E1 -23005.007,E2 -23005.007} C_VEL
LIN {X 0,Y 212.266,Z 442.2,A -85,B 0,C 180,E1 -23006.041,E2 -23006.041} C_VEL
LIN {X 0,Y 213.851,Z 430.247,A -85,B 0,C 180,E1 -23006.681,E2 -23006.681} C_VEL
LIN {X 0,Y 216.574,Z 393.278,A -85,B 0,C 180,E1 -23007.799,E2 -23007.799} C_VEL
LIN {X 0,Y 211.93,Z 383.375,A -85,B 0,C 180,E1 -23009.861,E2 -23009.861} C_VEL
LIN {X 0,Y 206.862,Z 374.909,A -85,B 0,C 180,E1 -23012.206,E2 -23012.206} C_VEL
LIN {X 0,Y 202.105,Z 367.566,A -85,B 0,C 180,E1 -23014.615,E2 -23014.615} C_VEL
LIN {X 0,Y 197.216,Z 360.532,A -85,B 0,C 180,E1 -23017.36,E2 -23017.36} C_VEL
LIN {X 0,Y 193.7,Z 355.836,A -85,B 0,C 180,E1 -23019.56,E2 -23019.56} C_VEL
LIN {X 0,Y 190.929,Z 352.087,A -85,B 0,C 180,E1 -23021.495,E2 -23021.495} C_VEL
LIN {X 0,Y 187.653,Z 348.243,A -85,B 0,C 180,E1 -23024.009,E2 -23024.009} C_VEL
LIN {X 0,Y 186.514,Z 346.378,A -85,B 0,C 180,E1 -23025.021,E2 -23025.021} C_VEL
LIN {X 0,Y 183.814,Z 343.91,A -85,B 0,C 180,E1 -23027.449,E2 -23027.449} C_VEL
LIN {X 0,Y 182.351,Z 340.956,A -85,B 0,C 180,E1 -23029.136,E2 -23029.136} C_VEL
LIN {X 0,Y 179.387,Z 338.829,A -85,B 0,C 180,E1 -23032.685,E2 -23032.685} C_VEL
LIN {X 0,Y 177.765,Z 335.926,A -85,B 0,C 180,E1 -23035.465,E2 -23035.465} C_VEL
LIN {X 0,Y 177.518,Z 335.138,A -85,B 0,C 180,E1 -23036.027,E2 -23036.027} C_VEL
LIN {X 0,Y 175,Z 333.921,A -85,B 0,C 180,E1 -23042.301,E2 -23042.301} C_VEL
LIN {X 0,Y 174.63,Z 333.814,A -85,B 0,C 180,E1 -23049.264,E2 -23049.264} C_VEL
LIN {X 0,Y 177.395,Z 335.417,A -85,B 0,C 180,E1 -23057.36,E2 -23057.36} C_VEL
LIN {X 0,Y 178.475,Z 338.156,A -85,B 0,C 180,E1 -23059.539,E2 -23059.539} C_VEL
LIN {X 0,Y 180.678,Z 340.327,A -85,B 0,C 180,E1 -23062.589,E2 -23062.589} C_VEL
LIN {X 0,Y 181.94,Z 341.507,A -85,B 0,C 180,E1 -23064.07,E2 -23064.07} C_VEL
LIN {X 0,Y 183.124,Z 343.092,A -85,B 0,C 180,E1 -23065.389,E2 -23065.389} C_VEL
LIN {X 0,Y 187.898,Z 349.6,A -85,B 0,C 180,E1 -23069.834,E2 -23069.834} C_VEL
LIN {X 0,Y 192.191,Z 355.947,A -85,B 0,C 180,E1 -23073.124,E2 -23073.124} C_VEL
LIN {X 0,Y 195.873,Z 361.796,A -85,B 0,C 180,E1 -23075.592,E2 -23075.592} C_VEL
LIN {X 0,Y 199.294,Z 367.498,A -85,B 0,C 180,E1 -23077.658,E2 -23077.658} C_VEL
LIN {X 0,Y 203.678,Z 375.09,A -85,B 0,C 180,E1 -23080.068,E2 -23080.068} C_VEL
LIN {X 0,Y 209.315,Z 386.294,A -85,B 0,C 180,E1 -23082.912,E2 -23082.912} C_VEL
LIN {X 0,Y 214.295,Z 397.805,A -85,B 0,C 180,E1 -23085.247,E2 -23085.247} C_VEL
LIN {X 0,Y 216.016,Z 402.234,A -85,B 0,C 180,E1 -23086.02,E2 -23086.02} C_VEL
LIN {X 0,Y 213.241,Z 441.068,A -85,B 0,C 180,E1 -23087.222,E2 -23087.222} C_VEL
LIN {X 0,Y 211.265,Z 454.56,A -85,B 0,C 180,E1 -23087.928,E2 -23087.928} C_VEL
LIN {X 0,Y 208.471,Z 467.194,A -85,B 0,C 180,E1 -23088.898,E2 -23088.898} C_VEL
LIN {X 0,Y 205.275,Z 478.185,A -85,B 0,C 180,E1 -23090.062,E2 -23090.062} C_VEL
LIN {X 0,Y 201.138,Z 489.679,A -85,B 0,C 180,E1 -23091.668,E2 -23091.668} C_VEL
LIN {X 0,Y 196.629,Z 500.547,A -85,B 0,C 180,E1 -23093.698,E2 -23093.698} C_VEL
LIN {X 0,Y 194.02,Z 504.978,A -85,B 0,C 180,E1 -23094.557,E2 -23094.557} C_VEL
LIN {X 0,Y 188.195,Z 511.814,A -85,B 0,C 180,E1 -23095.826,E2 -23095.826} C_VEL
LIN {X 0,Y 182.254,Z 518.072,A -85,B 0,C 180,E1 -23097.332,E2 -23097.332} C_VEL
LIN {X 0,Y 179.518,Z 521.568,A -85,B 0,C 180,E1 -23098.559,E2 -23098.559} C_VEL
LIN {X 0,Y 174.82,Z 528.813,A -85,B 0,C 180,E1 -23101.997,E2 -23101.997} C_VEL
LIN {X 0,Y 170.76,Z 534.586,A -85,B 0,C 180,E1 -23105.695,E2 -23105.695} C_VEL
LIN {X 0,Y 167.687,Z 538.56,A -85,B 0,C 180,E1 -23109.128,E2 -23109.128} C_VEL
LIN {X 0,Y 165.163,Z 541.521,A -85,B 0,C 180,E1 -23112.669,E2 -23112.669} C_VEL
LIN {X 0,Y 163.102,Z 544.002,A -85,B 0,C 180,E1 -23117.556,E2 -23117.556} C_VEL
LIN {X 0,Y 162.028,Z 544.954,A -85,B 0,C 180,E1 -23122.521,E2 -23122.521} C_VEL
LIN {X 0,Y 161.874,Z 544.471,A -85,B 0,C 180,E1 -23126.95,E2 -23126.95} C_VEL
LIN {X 0,Y 162.081,Z 543.385,A -85,B 0,C 180,E1 -23129.998,E2 -23129.998} C_VEL
LIN {X 0,Y 161.912,Z 541.496,A -85,B 0,C 180,E1 -23133.296,E2 -23133.296} C_VEL
LIN {X 0,Y 162.109,Z 537.977,A -85,B 0,C 180,E1 -23137.471,E2 -23137.471} C_VEL
LIN {X 0,Y 162.638,Z 533.666,A -85,B 0,C 180,E1 -23141.211,E2 -23141.211} C_VEL
LIN {X 0,Y 163.918,Z 527.112,A -85,B 0,C 180,E1 -23145.541,E2 -23145.541} C_VEL
LIN {X 0,Y 165.761,Z 519.898,A -85,B 0,C 180,E1 -23149.181,E2 -23149.181} C_VEL
LIN {X 0,Y 167.691,Z 512.539,A -85,B 0,C 180,E1 -23152.158,E2 -23152.158} C_VEL
LIN {X 0,Y 169.126,Z 507.036,A -85,B 0,C 180,E1 -23154.026,E2 -23154.026} C_VEL
LIN {X 0,Y 171.602,Z 497.305,A -85,B 0,C 180,E1 -23156.774,E2 -23156.774} C_VEL
LIN {X 0,Y 173.987,Z 487.333,A -85,B 0,C 180,E1 -23158.992,E2 -23158.992} C_VEL
LIN {X 0,Y 176.478,Z 476.519,A -85,B 0,C 180,E1 -23160.843,E2 -23160.843} C_VEL
LIN {X 0,Y 178.589,Z 464.554,A -85,B 0,C 180,E1 -23162.422,E2 -23162.422} C_VEL
LIN {X 0,Y 180.412,Z 451.671,A -85,B 0,C 180,E1 -23163.632,E2 -23163.632} C_VEL
LIN {X 0,Y 181.526,Z 439.035,A -85,B 0,C 180,E1 -23164.401,E2 -23164.401} C_VEL
LIN {X 0,Y 183.633,Z 392.72,A -85,B 0,C 180,E1 -23166.138,E2 -23166.138} C_VEL
LIN {X 0,Y 181.519,Z 370.724,A -85,B 0,C 180,E1 -23167.533,E2 -23167.533} C_VEL
LIN {X 0,Y 175.908,Z 355.493,A -85,B 0,C 180,E1 -23169.393,E2 -23169.393} C_VEL
LIN {X 0,Y 170.293,Z 342.909,A -85,B 0,C 180,E1 -23171.285,E2 -23171.285} C_VEL
LIN {X 0,Y 166.341,Z 335.181,A -85,B 0,C 180,E1 -23172.655,E2 -23172.655} C_VEL
LIN {X 0,Y 164.761,Z 331.717,A -85,B 0,C 180,E1 -23173.296,E2 -23173.296} C_VEL
LIN {X 0,Y 164.321,Z 330.016,A -85,B 0,C 180,E1 -23174.463,E2 -23174.463} C_VEL
LIN {X 0,Y 164.301,Z 330.008,A -85,B 0,C 180,E1 -23180.346,E2 -23180.346} C_VEL
LIN {X 0,Y 164.338,Z 330.01,A -85,B 0,C 180,E1 -23184.341,E2 -23184.341} C_VEL
LIN {X 0,Y 164.4,Z 330.006,A -85,B 0,C 180,E1 -23189.137,E2 -23189.137} C_VEL
LIN {X 0,Y 164.411,Z 330.002,A -85,B 0,C 180,E1 -23194.693,E2 -23194.693} C_VEL
LIN {X 0,Y 164.479,Z 329.988,A -85,B 0,C 180,E1 -23200.05,E2 -23200.05} C_VEL
LIN {X 0,Y 164.529,Z 329.976,A -85,B 0,C 180,E1 -23205.15,E2 -23205.15} C_VEL
LIN {X 0,Y 164.802,Z 329.95,A -85,B 0,C 180,E1 -23210.179,E2 -23210.179} C_VEL
LIN {X 0,Y 164.844,Z 329.922,A -85,B 0,C 180,E1 -23212.652,E2 -23212.652} C_VEL
LIN {X 0,Y 165.042,Z 329.917,A -85,B 0,C 180,E1 -23217.56,E2 -23217.56} C_VEL
LIN {X 0,Y 165.288,Z 329.894,A -85,B 0,C 180,E1 -23220,E2 -23220} C_VEL
LIN {X 0,Y 164.749,Z 329.93,A -85,B 0,C 180,E1 -23224.894,E2 -23224.894} C_VEL
LIN {X 0,Y 164.818,Z 329.922,A -85,B 0,C 180,E1 -23227.35,E2 -23227.35} C_VEL
LIN {X 0,Y 164.696,Z 329.966,A -85,B 0,C 180,E1 -23231.06,E2 -23231.06} C_VEL
LIN {X 0,Y 164.477,Z 329.994,A -85,B 0,C 180,E1 -23237.404,E2 -23237.404} C_VEL
LIN {X 0,Y 164.467,Z 329.996,A -85,B 0,C 180,E1 -23239.99,E2 -23239.99} C_VEL
LIN {X 0,Y 164.38,Z 330.006,A -85,B 0,C 180,E1 -23246.129,E2 -23246.129} C_VEL
LIN {X 0,Y 164.384,Z 330.006,A -85,B 0,C 180,E1 -23251.237,E2 -23251.237} C_VEL
LIN {X 0,Y 164.275,Z 330.02,A -85,B 0,C 180,E1 -23256.795,E2 -23256.795} C_VEL
LIN {X 0,Y 164.281,Z 330.014,A -85,B 0,C 180,E1 -23259.92,E2 -23259.92} C_VEL
LIN {X 0,Y 164.275,Z 330.015,A -85,B 0,C 180,E1 -23263.344,E2 -23263.344} C_VEL
LIN {X 0,Y 164.256,Z 330.025,A -85,B 0,C 180,E1 -23266.8,E2 -23266.8} C_VEL
LIN {X 0,Y 164.285,Z 330.019,A -85,B 0,C 180,E1 -23270.357,E2 -23270.357} C_VEL
LIN {X 0,Y 164.323,Z 330.015,A -85,B 0,C 180,E1 -23274.353,E2 -23274.353} C_VEL
LIN {X 0,Y 164.37,Z 330.006,A -85,B 0,C 180,E1 -23280.338,E2 -23280.338} C_VEL
LIN {X 0,Y 164.383,Z 330.203,A -85,B 0,C 180,E1 -23281.174,E2 -23281.174} C_VEL
LIN {X 0,Y 165.382,Z 332.88,A -85,B 0,C 180,E1 -23281.58,E2 -23281.58} C_VEL
LIN {X 0,Y 166.979,Z 335.279,A -85,B 0,C 180,E1 -23282.114,E2 -23282.114} C_VEL
LIN {X 0,Y 173.234,Z 345.843,A -85,B 0,C 180,E1 -23284.145,E2 -23284.145} C_VEL
LIN {X 0,Y 181.527,Z 362.419,A -85,B 0,C 180,E1 -23286.688,E2 -23286.688} C_VEL
LIN {X 0,Y 184.604,Z 370.479,A -85,B 0,C 180,E1 -23287.643,E2 -23287.643} C_VEL
LIN {X 0,Y 181.753,Z 428.507,A -85,B 0,C 180,E1 -23289.784,E2 -23289.784} C_VEL
LIN {X 0,Y 180.538,Z 441.919,A -85,B 0,C 180,E1 -23290.679,E2 -23290.679} C_VEL
LIN {X 0,Y 178.704,Z 454.775,A -85,B 0,C 180,E1 -23291.961,E2 -23291.961} C_VEL
LIN {X 0,Y 176.784,Z 466.14,A -85,B 0,C 180,E1 -23293.548,E2 -23293.548} C_VEL
LIN {X 0,Y 174.501,Z 477.802,A -85,B 0,C 180,E1 -23295.721,E2 -23295.721} C_VEL
LIN {X 0,Y 171.893,Z 488.349,A -85,B 0,C 180,E1 -23298.206,E2 -23298.206} C_VEL
LIN {X 0,Y 169.387,Z 497.839,A -85,B 0,C 180,E1 -23301.051,E2 -23301.051} C_VEL
LIN {X 0,Y 166.873,Z 506.968,A -85,B 0,C 180,E1 -23304.564,E2 -23304.564} C_VEL
LIN {X 0,Y 164.92,Z 514.324,A -85,B 0,C 180,E1 -23308.17,E2 -23308.17} C_VEL
LIN {X 0,Y 163.682,Z 519.305,A -85,B 0,C 180,E1 -23311.232,E2 -23311.232} C_VEL
LIN {X 0,Y 162.649,Z 524.146,A -85,B 0,C 180,E1 -23314.959,E2 -23314.959} C_VEL
LIN {X 0,Y 161.934,Z 527.875,A -85,B 0,C 180,E1 -23318.739,E2 -23318.739} C_VEL
LIN {X 0,Y 161.574,Z 530.576,A -85,B 0,C 180,E1 -23322.563,E2 -23322.563} C_VEL
LIN {X 0,Y 161.809,Z 532.544,A -85,B 0,C 180,E1 -23327.147,E2 -23327.147} C_VEL
LIN {X 0,Y 162.246,Z 533.085,A -85,B 0,C 180,E1 -23330.277,E2 -23330.277} C_VEL
LIN {X 0,Y 162.922,Z 533.092,A -85,B 0,C 180,E1 -23332.846,E2 -23332.846} C_VEL
LIN {X 0,Y 164.074,Z 532.53,A -85,B 0,C 180,E1 -23335.904,E2 -23335.904} C_VEL
LIN {X 0,Y 166.428,Z 530.519,A -85,B 0,C 180,E1 -23340.449,E2 -23340.449} C_VEL
LIN {X 0,Y 168.634,Z 528.254,A -85,B 0,C 180,E1 -23343.537,E2 -23343.537} C_VEL
LIN {X 0,Y 172.369,Z 523.825,A -85,B 0,C 180,E1 -23347.707,E2 -23347.707} C_VEL
LIN {X 0,Y 176.344,Z 518.603,A -85,B 0,C 180,E1 -23351.2,E2 -23351.2} C_VEL
LIN {X 0,Y 180.678,Z 512.164,A -85,B 0,C 180,E1 -23354.441,E2 -23354.441} C_VEL
LIN {X 0,Y 185.741,Z 503.895,A -85,B 0,C 180,E1 -23357.547,E2 -23357.547} C_VEL
LIN {X 0,Y 190.317,Z 495.375,A -85,B 0,C 180,E1 -23360.02,E2 -23360.02} C_VEL
LIN {X 0,Y 194.961,Z 485.604,A -85,B 0,C 180,E1 -23362.206,E2 -23362.206} C_VEL
LIN {X 0,Y 198.816,Z 475.716,A -85,B 0,C 180,E1 -23363.962,E2 -23363.962} C_VEL
LIN {X 0,Y 202.522,Z 464.397,A -85,B 0,C 180,E1 -23365.507,E2 -23365.507} C_VEL
LIN {X 0,Y 205.497,Z 453.029,A -85,B 0,C 180,E1 -23366.679,E2 -23366.679} C_VEL
LIN {X 0,Y 207.967,Z 440.048,A -85,B 0,C 180,E1 -23367.657,E2 -23367.657} C_VEL
LIN {X 0,Y 209.442,Z 428.469,A -85,B 0,C 180,E1 -23368.217,E2 -23368.217} C_VEL
LIN {X 0,Y 211.824,Z 395.737,A -85,B 0,C 180,E1 -23369.223,E2 -23369.223} C_VEL
LIN {X 0,Y 207.306,Z 386.371,A -85,B 0,C 180,E1 -23371.363,E2 -23371.363} C_VEL
LIN {X 0,Y 200.982,Z 375.863,A -85,B 0,C 180,E1 -23374.567,E2 -23374.567} C_VEL
LIN {X 0,Y 196.354,Z 369.008,A -85,B 0,C 180,E1 -23377.184,E2 -23377.184} C_VEL
LIN {X 0,Y 191.616,Z 362.234,A -85,B 0,C 180,E1 -23380.237,E2 -23380.237} C_VEL
LIN {X 0,Y 188.177,Z 357.667,A -85,B 0,C 180,E1 -23382.773,E2 -23382.773} C_VEL
LIN {X 0,Y 185.636,Z 354.447,A -85,B 0,C 180,E1 -23384.869,E2 -23384.869} C_VEL
LIN {X 0,Y 184.778,Z 353.032,A -85,B 0,C 180,E1 -23385.669,E2 -23385.669} C_VEL
LIN {X 0,Y 182.066,Z 350.291,A -85,B 0,C 180,E1 -23388.255,E2 -23388.255} C_VEL
LIN {X 0,Y 180.803,Z 347.798,A -85,B 0,C 180,E1 -23389.778,E2 -23389.778} C_VEL
LIN {X 0,Y 177.604,Z 344.972,A -85,B 0,C 180,E1 -23393.984,E2 -23393.984} C_VEL
LIN {X 0,Y 176.308,Z 342.094,A -85,B 0,C 180,E1 -23396.572,E2 -23396.572} C_VEL
LIN {X 0,Y 174.117,Z 340.967,A -85,B 0,C 180,E1 -23402.313,E2 -23402.313} C_VEL
LIN {X 0,Y 173.587,Z 340.702,A -85,B 0,C 180,E1 -23406.976,E2 -23406.976} C_VEL
LIN {X 0,Y 174.501,Z 341.539,A -85,B 0,C 180,E1 -23412.798,E2 -23412.798} C_VEL
LIN {X 0,Y 176.192,Z 342.283,A -85,B 0,C 180,E1 -23416.797,E2 -23416.797} C_VEL
LIN {X 0,Y 177.251,Z 344.99,A -85,B 0,C 180,E1 -23419.052,E2 -23419.052} C_VEL
LIN {X 0,Y 179.391,Z 347.19,A -85,B 0,C 180,E1 -23422.153,E2 -23422.153} C_VEL
LIN {X 0,Y 180.502,Z 348.229,A -85,B 0,C 180,E1 -23423.508,E2 -23423.508} C_VEL
LIN {X 0,Y 182.61,Z 351.271,A -85,B 0,C 180,E1 -23425.886,E2 -23425.886} C_VEL
LIN {X 0,Y 186.017,Z 356.094,A -85,B 0,C 180,E1 -23429.117,E2 -23429.117} C_VEL
LIN {X 0,Y 189.976,Z 362.148,A -85,B 0,C 180,E1 -23432.316,E2 -23432.316} C_VEL
LIN {X 0,Y 193.357,Z 367.753,A -85,B 0,C 180,E1 -23434.717,E2 -23434.717} C_VEL
LIN {X 0,Y 196.975,Z 374.031,A -85,B 0,C 180,E1 -23437.012,E2 -23437.012} C_VEL
LIN {X 0,Y 200.81,Z 380.979,A -85,B 0,C 180,E1 -23439.227,E2 -23439.227} C_VEL
LIN {X 0,Y 205.838,Z 391.294,A -85,B 0,C 180,E1 -23441.907,E2 -23441.907} C_VEL
LIN {X 0,Y 210.515,Z 402.613,A -85,B 0,C 180,E1 -23444.242,E2 -23444.242} C_VEL
LIN {X 0,Y 211.265,Z 404.551,A -85,B 0,C 180,E1 -23444.603,E2 -23444.603} C_VEL
LIN {X 0,Y 208.91,Z 438.039,A -85,B 0,C 180,E1 -23445.654,E2 -23445.654} C_VEL
LIN {X 0,Y 207.163,Z 451.046,A -85,B 0,C 180,E1 -23446.258,E2 -23446.258} C_VEL
LIN {X 0,Y 204.344,Z 464.31,A -85,B 0,C 180,E1 -23447.213,E2 -23447.213} C_VEL
LIN {X 0,Y 200.969,Z 475.95,A -85,B 0,C 180,E1 -23448.359,E2 -23448.359} C_VEL
LIN {X 0,Y 197.224,Z 486.575,A -85,B 0,C 180,E1 -23449.767,E2 -23449.767} C_VEL
LIN {X 0,Y 192.641,Z 497.453,A -85,B 0,C 180,E1 -23451.668,E2 -23451.668} C_VEL
LIN {X 0,Y 187.882,Z 507.216,A -85,B 0,C 180,E1 -23453.902,E2 -23453.902} C_VEL
LIN {X 0,Y 183.397,Z 515.248,A -85,B 0,C 180,E1 -23456.243,E2 -23456.243} C_VEL
LIN {X 0,Y 179.518,Z 521.568,A -85,B 0,C 180,E1 -23458.559,E2 -23458.559} C_VEL
LIN {X 0,Y 176.827,Z 524.886,A -85,B 0,C 180,E1 -23459.882,E2 -23459.882} C_VEL
LIN {X 0,Y 171.012,Z 529.834,A -85,B 0,C 180,E1 -23461.971,E2 -23461.971} C_VEL
LIN {X 0,Y 165.335,Z 534.088,A -85,B 0,C 180,E1 -23464.326,E2 -23464.326} C_VEL
LIN {X 0,Y 162.928,Z 536.27,A -85,B 0,C 180,E1 -23466.047,E2 -23466.047} C_VEL
LIN {X 0,Y 160.091,Z 539.589,A -85,B 0,C 180,E1 -23469.438,E2 -23469.438} C_VEL
LIN {X 0,Y 158.384,Z 541.413,A -85,B 0,C 180,E1 -23471.902,E2 -23471.902} C_VEL
LIN {X 0,Y 156.129,Z 543.817,A -85,B 0,C 180,E1 -23476.991,E2 -23476.991} C_VEL
LIN {X 0,Y 154.972,Z 544.692,A -85,B 0,C 180,E1 -23482.179,E2 -23482.179} C_VEL
LIN {X 0,Y 154.814,Z 544.041,A -85,B 0,C 180,E1 -23487.104,E2 -23487.104} C_VEL
LIN {X 0,Y 154.986,Z 543.006,A -85,B 0,C 180,E1 -23489.998,E2 -23489.998} C_VEL
LIN {X 0,Y 154.832,Z 541.341,A -85,B 0,C 180,E1 -23493.024,E2 -23493.024} C_VEL
LIN {X 0,Y 155.035,Z 537.458,A -85,B 0,C 180,E1 -23497.814,E2 -23497.814} C_VEL
LIN {X 0,Y 155.62,Z 533.07,A -85,B 0,C 180,E1 -23501.724,E2 -23501.724} C_VEL
LIN {X 0,Y 156.754,Z 527.456,A -85,B 0,C 180,E1 -23505.603,E2 -23505.603} C_VEL
LIN {X 0,Y 158.677,Z 520.444,A -85,B 0,C 180,E1 -23509.399,E2 -23509.399} C_VEL
LIN {X 0,Y 160.679,Z 513.252,A -85,B 0,C 180,E1 -23512.5,E2 -23512.5} C_VEL
LIN {X 0,Y 161.912,Z 508.372,A -85,B 0,C 180,E1 -23514.282,E2 -23514.282} C_VEL
LIN {X 0,Y 164.379,Z 499.411,A -85,B 0,C 180,E1 -23517.016,E2 -23517.016} C_VEL
LIN {X 0,Y 167.167,Z 488.663,A -85,B 0,C 180,E1 -23519.601,E2 -23519.601} C_VEL
LIN {X 0,Y 169.603,Z 478.275,A -85,B 0,C 180,E1 -23521.542,E2 -23521.542} C_VEL
LIN {X 0,Y 172.03,Z 465.846,A -85,B 0,C 180,E1 -23523.294,E2 -23523.294} C_VEL
LIN {X 0,Y 173.85,Z 453.568,A -85,B 0,C 180,E1 -23524.545,E2 -23524.545} C_VEL
LIN {X 0,Y 175.183,Z 440.764,A -85,B 0,C 180,E1 -23525.415,E2 -23525.415} C_VEL
LIN {X 0,Y 177.558,Z 394.417,A -85,B 0,C 180,E1 -23527.199,E2 -23527.199} C_VEL
LIN {X 0,Y 175.646,Z 372.992,A -85,B 0,C 180,E1 -23528.603,E2 -23528.603} C_VEL
LIN {X 0,Y 170.046,Z 357.762,A -85,B 0,C 180,E1 -23530.585,E2 -23530.585} C_VEL
LIN {X 0,Y 164.055,Z 344.322,A -85,B 0,C 180,E1 -23532.749,E2 -23532.749} C_VEL
LIN {X 0,Y 158.997,Z 334.72,A -85,B 0,C 180,E1 -23534.653,E2 -23534.653} C_VEL
LIN {X 0,Y 157.536,Z 332.224,A -85,B 0,C 180,E1 -23535.219,E2 -23535.219} C_VEL
LIN {X 0,Y 157.319,Z 331.344,A -85,B 0,C 180,E1 -23535.406,E2 -23535.406} C_VEL
LIN {X 0,Y 157.226,Z 330.901,A -85,B 0,C 180,E1 -23535.861,E2 -23535.861} C_VEL
LIN {X 0,Y 157.233,Z 330.891,A -85,B 0,C 180,E1 -23541.261,E2 -23541.261} C_VEL
LIN {X 0,Y 157.286,Z 330.889,A -85,B 0,C 180,E1 -23544.488,E2 -23544.488} C_VEL
LIN {X 0,Y 157.297,Z 330.886,A -85,B 0,C 180,E1 -23548.089,E2 -23548.089} C_VEL
LIN {X 0,Y 157.317,Z 330.888,A -85,B 0,C 180,E1 -23553.465,E2 -23553.465} C_VEL
LIN {X 0,Y 157.388,Z 330.874,A -85,B 0,C 180,E1 -23559.667,E2 -23559.667} C_VEL
LIN {X 0,Y 157.454,Z 330.85,A -85,B 0,C 180,E1 -23564.466,E2 -23564.466} C_VEL
LIN {X 0,Y 157.728,Z 330.832,A -85,B 0,C 180,E1 -23569.733,E2 -23569.733} C_VEL
LIN {X 0,Y 157.802,Z 330.801,A -85,B 0,C 180,E1 -23572.322,E2 -23572.322} C_VEL
LIN {X 0,Y 158.25,Z 330.771,A -85,B 0,C 180,E1 -23580,E2 -23580} C_VEL
LIN {X 0,Y 157.756,Z 330.803,A -85,B 0,C 180,E1 -23587.681,E2 -23587.681} C_VEL
LIN {X 0,Y 157.63,Z 330.847,A -85,B 0,C 180,E1 -23591.236,E2 -23591.236} C_VEL
LIN {X 0,Y 157.435,Z 330.864,A -85,B 0,C 180,E1 -23595.536,E2 -23595.536} C_VEL
LIN {X 0,Y 157.362,Z 330.876,A -85,B 0,C 180,E1 -23600.934,E2 -23600.934} C_VEL
LIN {X 0,Y 157.304,Z 330.884,A -85,B 0,C 180,E1 -23606.682,E2 -23606.682} C_VEL
LIN {X 0,Y 157.276,Z 330.887,A -85,B 0,C 180,E1 -23612.428,E2 -23612.428} C_VEL
LIN {X 0,Y 157.254,Z 330.895,A -85,B 0,C 180,E1 -23616.446,E2 -23616.446} C_VEL
LIN {X 0,Y 157.185,Z 330.903,A -85,B 0,C 180,E1 -23622.12,E2 -23622.12} C_VEL
LIN {X 0,Y 157.186,Z 330.901,A -85,B 0,C 180,E1 -23627.884,E2 -23627.884} C_VEL
LIN {X 0,Y 157.255,Z 330.892,A -85,B 0,C 180,E1 -23633.558,E2 -23633.558} C_VEL
LIN {X 0,Y 157.344,Z 330.885,A -85,B 0,C 180,E1 -23639.217,E2 -23639.217} C_VEL
LIN {X 0,Y 158.409,Z 333.879,A -85,B 0,C 180,E1 -23639.736,E2 -23639.736} C_VEL
LIN {X 0,Y 159.998,Z 336.027,A -85,B 0,C 180,E1 -23640.309,E2 -23640.309} C_VEL
LIN {X 0,Y 168.332,Z 350.166,A -85,B 0,C 180,E1 -23643.226,E2 -23643.226} C_VEL
LIN {X 0,Y 176.47,Z 366.745,A -85,B 0,C 180,E1 -23645.871,E2 -23645.871} C_VEL
LIN {X 0,Y 178.433,Z 372.091,A -85,B 0,C 180,E1 -23646.527,E2 -23646.527} C_VEL
LIN {X 0,Y 177.232,Z 398.377,A -85,B 0,C 180,E1 -23647.527,E2 -23647.527} C_VEL
LIN {X 0,Y 175.399,Z 430.625,A -85,B 0,C 180,E1 -23648.784,E2 -23648.784} C_VEL
LIN {X 0,Y 174.091,Z 444.154,A -85,B 0,C 180,E1 -23649.78,E2 -23649.78} C_VEL
LIN {X 0,Y 172.138,Z 456.468,A -85,B 0,C 180,E1 -23651.093,E2 -23651.093} C_VEL
LIN {X 0,Y 170.011,Z 468.237,A -85,B 0,C 180,E1 -23652.872,E2 -23652.872} C_VEL
LIN {X 0,Y 167.638,Z 479.56,A -85,B 0,C 180,E1 -23655.123,E2 -23655.123} C_VEL
LIN {X 0,Y 164.952,Z 489.833,A -85,B 0,C 180,E1 -23657.702,E2 -23657.702} C_VEL
LIN {X 0,Y 162.364,Z 499.05,A -85,B 0,C 180,E1 -23660.66,E2 -23660.66} C_VEL
LIN {X 0,Y 159.789,Z 508.019,A -85,B 0,C 180,E1 -23664.323,E2 -23664.323} C_VEL
LIN {X 0,Y 157.796,Z 515.23,A -85,B 0,C 180,E1 -23668.088,E2 -23668.088} C_VEL
LIN {X 0,Y 156.536,Z 520.098,A -85,B 0,C 180,E1 -23671.288,E2 -23671.288} C_VEL
LIN {X 0,Y 155.379,Z 525.342,A -85,B 0,C 180,E1 -23675.675,E2 -23675.675} C_VEL
LIN {X 0,Y 154.596,Z 529.424,A -85,B 0,C 180,E1 -23680.479,E2 -23680.479} C_VEL
LIN {X 0,Y 154.477,Z 531.062,A -85,B 0,C 180,E1 -23683.15,E2 -23683.15} C_VEL
LIN {X 0,Y 154.744,Z 532.791,A -85,B 0,C 180,E1 -23687.491,E2 -23687.491} C_VEL
LIN {X 0,Y 155.34,Z 533.383,A -85,B 0,C 180,E1 -23691.221,E2 -23691.221} C_VEL
LIN {X 0,Y 156.134,Z 533.341,A -85,B 0,C 180,E1 -23693.9,E2 -23693.9} C_VEL
LIN {X 0,Y 157.225,Z 532.822,A -85,B 0,C 180,E1 -23696.618,E2 -23696.618} C_VEL
LIN {X 0,Y 158.47,Z 531.915,A -85,B 0,C 180,E1 -23699.2,E2 -23699.2} C_VEL
LIN {X 0,Y 160.055,Z 530.574,A -85,B 0,C 180,E1 -23701.799,E2 -23701.799} C_VEL
LIN {X 0,Y 162.893,Z 527.786,A -85,B 0,C 180,E1 -23705.473,E2 -23705.473} C_VEL
LIN {X 0,Y 166.545,Z 523.668,A -85,B 0,C 180,E1 -23709.272,E2 -23709.272} C_VEL
LIN {X 0,Y 171.457,Z 517.375,A -85,B 0,C 180,E1 -23713.361,E2 -23713.361} C_VEL
LIN {X 0,Y 176.201,Z 510.571,A -85,B 0,C 180,E1 -23716.619,E2 -23716.619} C_VEL
LIN {X 0,Y 180.807,Z 503.277,A -85,B 0,C 180,E1 -23719.287,E2 -23719.287} C_VEL
LIN {X 0,Y 185.645,Z 494.585,A -85,B 0,C 180,E1 -23721.772,E2 -23721.772} C_VEL
LIN {X 0,Y 190.825,Z 483.726,A -85,B 0,C 180,E1 -23724.122,E2 -23724.122} C_VEL
LIN {X 0,Y 195.104,Z 472.845,A -85,B 0,C 180,E1 -23725.947,E2 -23725.947} C_VEL
LIN {X 0,Y 198.977,Z 460.612,A -85,B 0,C 180,E1 -23727.49,E2 -23727.49} C_VEL
LIN {X 0,Y 202.003,Z 448.356,A -85,B 0,C 180,E1 -23728.602,E2 -23728.602} C_VEL
LIN {X 0,Y 204.07,Z 436.028,A -85,B 0,C 180,E1 -23729.428,E2 -23729.428} C_VEL
LIN {X 0,Y 205.51,Z 422.387,A -85,B 0,C 180,E1 -23729.955,E2 -23729.955} C_VEL
LIN {X 0,Y 207.286,Z 398.502,A -85,B 0,C 180,E1 -23730.671,E2 -23730.671} C_VEL
LIN {X 0,Y 203.827,Z 391.331,A -85,B 0,C 180,E1 -23732.412,E2 -23732.412} C_VEL
LIN {X 0,Y 197.948,Z 381.236,A -85,B 0,C 180,E1 -23735.571,E2 -23735.571} C_VEL
LIN {X 0,Y 192.278,Z 372.602,A -85,B 0,C 180,E1 -23739.034,E2 -23739.034} C_VEL
LIN {X 0,Y 189.041,Z 368.044,A -85,B 0,C 180,E1 -23741.303,E2 -23741.303} C_VEL
LIN {X 0,Y 186.19,Z 364.048,A -85,B 0,C 180,E1 -23743.537,E2 -23743.537} C_VEL
LIN {X 0,Y 183.555,Z 360.447,A -85,B 0,C 180,E1 -23745.854,E2 -23745.854} C_VEL
LIN {X 0,Y 182.962,Z 359.558,A -85,B 0,C 180,E1 -23746.427,E2 -23746.427} C_VEL
LIN {X 0,Y 180.339,Z 356.656,A -85,B 0,C 180,E1 -23749.093,E2 -23749.093} C_VEL
LIN {X 0,Y 179.04,Z 354.373,A -85,B 0,C 180,E1 -23750.727,E2 -23750.727} C_VEL
LIN {X 0,Y 176.214,Z 351.543,A -85,B 0,C 180,E1 -23754.766,E2 -23754.766} C_VEL
LIN {X 0,Y 175.193,Z 349.104,A -85,B 0,C 180,E1 -23756.967,E2 -23756.967} C_VEL
LIN {X 0,Y 173.236,Z 347.998,A -85,B 0,C 180,E1 -23762.325,E2 -23762.325} C_VEL
LIN {X 0,Y 172.885,Z 347.928,A -85,B 0,C 180,E1 -23769.358,E2 -23769.358} C_VEL
LIN {X 0,Y 175.037,Z 349.312,A -85,B 0,C 180,E1 -23776.323,E2 -23776.323} C_VEL
LIN {X 0,Y 176.373,Z 352.331,A -85,B 0,C 180,E1 -23779.151,E2 -23779.151} C_VEL
LIN {X 0,Y 179.203,Z 355.106,A -85,B 0,C 180,E1 -23783.09,E2 -23783.09} C_VEL
LIN {X 0,Y 184,Z 362.261,A -85,B 0,C 180,E1 -23788.224,E2 -23788.224} C_VEL
LIN {X 0,Y 187.846,Z 368.464,A -85,B 0,C 180,E1 -23791.52,E2 -23791.52} C_VEL
LIN {X 0,Y 191.189,Z 374.255,A -85,B 0,C 180,E1 -23794.027,E2 -23794.027} C_VEL
LIN {X 0,Y 194.149,Z 379.598,A -85,B 0,C 180,E1 -23796.014,E2 -23796.014} C_VEL
LIN {X 0,Y 197.688,Z 386.243,A -85,B 0,C 180,E1 -23798.185,E2 -23798.185} C_VEL
LIN {X 0,Y 202.194,Z 395.844,A -85,B 0,C 180,E1 -23800.746,E2 -23800.746} C_VEL
LIN {X 0,Y 206.592,Z 406.731,A -85,B 0,C 180,E1 -23803.084,E2 -23803.084} C_VEL
LIN {X 0,Y 206.766,Z 407.251,A -85,B 0,C 180,E1 -23803.177,E2 -23803.177} C_VEL
LIN {X 0,Y 204.134,Z 440.544,A -85,B 0,C 180,E1 -23804.215,E2 -23804.215} C_VEL
LIN {X 0,Y 202.031,Z 454.089,A -85,B 0,C 180,E1 -23804.935,E2 -23804.935} C_VEL
LIN {X 0,Y 199.251,Z 465.962,A -85,B 0,C 180,E1 -23805.842,E2 -23805.842} C_VEL
LIN {X 0,Y 195.766,Z 477.144,A -85,B 0,C 180,E1 -23806.991,E2 -23806.991} C_VEL
LIN {X 0,Y 191.324,Z 488.722,A -85,B 0,C 180,E1 -23808.607,E2 -23808.607} C_VEL
LIN {X 0,Y 186.644,Z 499.146,A -85,B 0,C 180,E1 -23810.547,E2 -23810.547} C_VEL
LIN {X 0,Y 182.226,Z 507.688,A -85,B 0,C 180,E1 -23812.594,E2 -23812.594} C_VEL
LIN {X 0,Y 177.557,Z 515.592,A -85,B 0,C 180,E1 -23814.974,E2 -23814.974} C_VEL
LIN {X 0,Y 172.469,Z 523.364,A -85,B 0,C 180,E1 -23818.01,E2 -23818.01} C_VEL
LIN {X 0,Y 168.091,Z 529.612,A -85,B 0,C 180,E1 -23821.261,E2 -23821.261} C_VEL
LIN {X 0,Y 164.312,Z 534.611,A -85,B 0,C 180,E1 -23824.675,E2 -23824.675} C_VEL
LIN {X 0,Y 162.928,Z 536.27,A -85,B 0,C 180,E1 -23826.047,E2 -23826.047} C_VEL
LIN {X 0,Y 160.619,Z 538.259,A -85,B 0,C 180,E1 -23827.853,E2 -23827.853} C_VEL
LIN {X 0,Y 155.466,Z 540.89,A -85,B 0,C 180,E1 -23830.78,E2 -23830.78} C_VEL
LIN {X 0,Y 150.782,Z 542.77,A -85,B 0,C 180,E1 -23833.961,E2 -23833.961} C_VEL
LIN {X 0,Y 149.264,Z 543.536,A -85,B 0,C 180,E1 -23836.107,E2 -23836.107} C_VEL
LIN {X 0,Y 148.418,Z 544.231,A -85,B 0,C 180,E1 -23839.08,E2 -23839.08} C_VEL
LIN {X 0,Y 147.748,Z 544.202,A -85,B 0,C 180,E1 -23844.539,E2 -23844.539} C_VEL
LIN {X 0,Y 147.756,Z 543.61,A -85,B 0,C 180,E1 -23847.272,E2 -23847.272} C_VEL
LIN {X 0,Y 147.892,Z 542.627,A -85,B 0,C 180,E1 -23849.998,E2 -23849.998} C_VEL
LIN {X 0,Y 147.755,Z 541.185,A -85,B 0,C 180,E1 -23852.724,E2 -23852.724} C_VEL
LIN {X 0,Y 147.858,Z 538.191,A -85,B 0,C 180,E1 -23856.822,E2 -23856.822} C_VEL
LIN {X 0,Y 148.367,Z 534.108,A -85,B 0,C 180,E1 -23860.92,E2 -23860.92} C_VEL
LIN {X 0,Y 149.616,Z 527.795,A -85,B 0,C 180,E1 -23865.668,E2 -23865.668} C_VEL
LIN {X 0,Y 151.58,Z 520.924,A -85,B 0,C 180,E1 -23869.64,E2 -23869.64} C_VEL
LIN {X 0,Y 153.655,Z 513.89,A -85,B 0,C 180,E1 -23872.876,E2 -23872.876} C_VEL
LIN {X 0,Y 155.099,Z 508.414,A -85,B 0,C 180,E1 -23875.006,E2 -23875.006} C_VEL
LIN {X 0,Y 157.734,Z 499.343,A -85,B 0,C 180,E1 -23877.892,E2 -23877.892} C_VEL
LIN {X 0,Y 160.643,Z 488.636,A -85,B 0,C 180,E1 -23880.567,E2 -23880.567} C_VEL
LIN {X 0,Y 163.179,Z 478.301,A -85,B 0,C 180,E1 -23882.57,E2 -23882.57} C_VEL
LIN {X 0,Y 165.702,Z 465.994,A -85,B 0,C 180,E1 -23884.374,E2 -23884.374} C_VEL
LIN {X 0,Y 167.601,Z 453.773,A -85,B 0,C 180,E1 -23885.668,E2 -23885.668} C_VEL
LIN {X 0,Y 169.006,Z 441.001,A -85,B 0,C 180,E1 -23886.573,E2 -23886.573} C_VEL
LIN {X 0,Y 171.181,Z 401.11,A -85,B 0,C 180,E1 -23888.165,E2 -23888.165} C_VEL
LIN {X 0,Y 171.444,Z 393.96,A -85,B 0,C 180,E1 -23888.462,E2 -23888.462} C_VEL
LIN {X 0,Y 169.836,Z 375.225,A -85,B 0,C 180,E1 -23889.748,E2 -23889.748} C_VEL
LIN {X 0,Y 164.127,Z 359.67,A -85,B 0,C 180,E1 -23891.905,E2 -23891.905} C_VEL
LIN {X 0,Y 158.735,Z 347.647,A -85,B 0,C 180,E1 -23893.989,E2 -23893.989} C_VEL
LIN {X 0,Y 154.365,Z 339.259,A -85,B 0,C 180,E1 -23895.752,E2 -23895.752} C_VEL
LIN {X 0,Y 152.279,Z 335.979,A -85,B 0,C 180,E1 -23896.601,E2 -23896.601} C_VEL
LIN {X 0,Y 150.556,Z 333.308,A -85,B 0,C 180,E1 -23897.326,E2 -23897.326} C_VEL
LIN {X 0,Y 150.175,Z 331.779,A -85,B 0,C 180,E1 -23897.603,E2 -23897.603} C_VEL
LIN {X 0,Y 150.211,Z 331.774,A -85,B 0,C 180,E1 -23902.688,E2 -23902.688} C_VEL
LIN {X 0,Y 150.218,Z 331.767,A -85,B 0,C 180,E1 -23907.361,E2 -23907.361} C_VEL
LIN {X 0,Y 150.24,Z 331.768,A -85,B 0,C 180,E1 -23912.716,E2 -23912.716} C_VEL
LIN {X 0,Y 150.345,Z 331.753,A -85,B 0,C 180,E1 -23919.207,E2 -23919.207} C_VEL
LIN {X 0,Y 150.36,Z 331.727,A -85,B 0,C 180,E1 -23923.713,E2 -23923.713} C_VEL
LIN {X 0,Y 150.652,Z 331.716,A -85,B 0,C 180,E1 -23929.246,E2 -23929.246} C_VEL
LIN {X 0,Y 150.738,Z 331.683,A -85,B 0,C 180,E1 -23931.96,E2 -23931.96} C_VEL
LIN {X 0,Y 151.21,Z 331.648,A -85,B 0,C 180,E1 -23940,E2 -23940} C_VEL
LIN {X 0,Y 150.678,Z 331.686,A -85,B 0,C 180,E1 -23948.044,E2 -23948.044} C_VEL
LIN {X 0,Y 150.57,Z 331.726,A -85,B 0,C 180,E1 -23951.437,E2 -23951.437} C_VEL
LIN {X 0,Y 150.347,Z 331.749,A -85,B 0,C 180,E1 -23956.289,E2 -23956.289} C_VEL
LIN {X 0,Y 150.344,Z 331.751,A -85,B 0,C 180,E1 -23960.792,E2 -23960.792} C_VEL
LIN {X 0,Y 150.237,Z 331.762,A -85,B 0,C 180,E1 -23967.282,E2 -23967.282} C_VEL
LIN {X 0,Y 150.215,Z 331.765,A -85,B 0,C 180,E1 -23972.637,E2 -23972.637} C_VEL
LIN {X 0,Y 150.164,Z 331.775,A -85,B 0,C 180,E1 -23977.476,E2 -23977.476} C_VEL
LIN {X 0,Y 150.128,Z 331.782,A -85,B 0,C 180,E1 -23981.499,E2 -23981.499} C_VEL
LIN {X 0,Y 150.122,Z 331.78,A -85,B 0,C 180,E1 -23985.397,E2 -23985.397} C_VEL
LIN {X 0,Y 150.132,Z 331.777,A -85,B 0,C 180,E1 -23989.056,E2 -23989.056} C_VEL
LIN {X 0,Y 150.172,Z 331.774,A -85,B 0,C 180,E1 -23992.712,E2 -23992.712} C_VEL
LIN {X 0,Y 150.195,Z 331.772,A -85,B 0,C 180,E1 -23997.056,E2 -23997.056} C_VEL
LIN {X 0,Y 151.223,Z 334.621,A -85,B 0,C 180,E1 -23997.583,E2 -23997.583} C_VEL
LIN {X 0,Y 153.076,Z 336.966,A -85,B 0,C 180,E1 -23998.319,E2 -23998.319} C_VEL
LIN {X 0,Y 161.545,Z 351.022,A -85,B 0,C 180,E1 -24001.569,E2 -24001.569} C_VEL
LIN {X 0,Y 168.56,Z 364.816,A -85,B 0,C 180,E1 -24004.034,E2 -24004.034} C_VEL
LIN {X 0,Y 172.412,Z 373.797,A -85,B 0,C 180,E1 -24005.352,E2 -24005.352} C_VEL
LIN {X 0,Y 169.374,Z 429.723,A -85,B 0,C 180,E1 -24007.537,E2 -24007.537} C_VEL
LIN {X 0,Y 167.994,Z 443.396,A -85,B 0,C 180,E1 -24008.53,E2 -24008.53} C_VEL
LIN {X 0,Y 165.986,Z 456.014,A -85,B 0,C 180,E1 -24009.88,E2 -24009.88} C_VEL
LIN {X 0,Y 163.901,Z 467.173,A -85,B 0,C 180,E1 -24011.567,E2 -24011.567} C_VEL
LIN {X 0,Y 161.41,Z 478.732,A -85,B 0,C 180,E1 -24013.887,E2 -24013.887} C_VEL
LIN {X 0,Y 158.557,Z 489.212,A -85,B 0,C 180,E1 -24016.545,E2 -24016.545} C_VEL
LIN {X 0,Y 155.832,Z 498.624,A -85,B 0,C 180,E1 -24019.609,E2 -24019.609} C_VEL
LIN {X 0,Y 153.08,Z 507.709,A -85,B 0,C 180,E1 -24023.411,E2 -24023.411} C_VEL
LIN {X 0,Y 150.924,Z 515.031,A -85,B 0,C 180,E1 -24027.333,E2 -24027.333} C_VEL
LIN {X 0,Y 149.378,Z 520.886,A -85,B 0,C 180,E1 -24031.35,E2 -24031.35} C_VEL
LIN {X 0,Y 148.291,Z 525.631,A -85,B 0,C 180,E1 -24035.579,E2 -24035.579} C_VEL
LIN {X 0,Y 147.621,Z 529.03,A -85,B 0,C 180,E1 -24039.594,E2 -24039.594} C_VEL
LIN {X 0,Y 147.403,Z 531.541,A -85,B 0,C 180,E1 -24043.794,E2 -24043.794} C_VEL
LIN {X 0,Y 147.702,Z 533.045,A -85,B 0,C 180,E1 -24047.889,E2 -24047.889} C_VEL
LIN {X 0,Y 148.485,Z 533.681,A -85,B 0,C 180,E1 -24052.252,E2 -24052.252} C_VEL
LIN {X 0,Y 150.41,Z 533.112,A -85,B 0,C 180,E1 -24057.403,E2 -24057.403} C_VEL
LIN {X 0,Y 152.031,Z 532.02,A -85,B 0,C 180,E1 -24060.566,E2 -24060.566} C_VEL
LIN {X 0,Y 153.797,Z 530.62,A -85,B 0,C 180,E1 -24063.256,E2 -24063.256} C_VEL
LIN {X 0,Y 157.002,Z 527.622,A -85,B 0,C 180,E1 -24067.181,E2 -24067.181} C_VEL
LIN {X 0,Y 160.851,Z 523.493,A -85,B 0,C 180,E1 -24070.951,E2 -24070.951} C_VEL
LIN {X 0,Y 166.135,Z 517.058,A -85,B 0,C 180,E1 -24075.121,E2 -24075.121} C_VEL
LIN {X 0,Y 170.383,Z 511.248,A -85,B 0,C 180,E1 -24077.944,E2 -24077.944} C_VEL
LIN {X 0,Y 176.041,Z 502.67,A -85,B 0,C 180,E1 -24081.124,E2 -24081.124} C_VEL
LIN {X 0,Y 181.706,Z 492.724,A -85,B 0,C 180,E1 -24083.845,E2 -24083.845} C_VEL
LIN {X 0,Y 186.566,Z 482.623,A -85,B 0,C 180,E1 -24085.972,E2 -24085.972} C_VEL
LIN {X 0,Y 191.037,Z 471.351,A -85,B 0,C 180,E1 -24087.796,E2 -24087.796} C_VEL
LIN {X 0,Y 194.823,Z 459.607,A -85,B 0,C 180,E1 -24089.207,E2 -24089.207} C_VEL
LIN {X 0,Y 197.855,Z 447.285,A -85,B 0,C 180,E1 -24090.304,E2 -24090.304} C_VEL
LIN {X 0,Y 199.933,Z 434.92,A -85,B 0,C 180,E1 -24091.085,E2 -24091.085} C_VEL
LIN {X 0,Y 201.605,Z 418.065,A -85,B 0,C 180,E1 -24091.672,E2 -24091.672} C_VEL
LIN {X 0,Y 202.851,Z 401.327,A -85,B 0,C 180,E1 -24092.193,E2 -24092.193} C_VEL
LIN {X 0,Y 199.824,Z 395.13,A -85,B 0,C 180,E1 -24093.823,E2 -24093.823} C_VEL
LIN {X 0,Y 194.207,Z 385.458,A -85,B 0,C 180,E1 -24097.067,E2 -24097.067} C_VEL
LIN {X 0,Y 189.631,Z 378.321,A -85,B 0,C 180,E1 -24100.083,E2 -24100.083} C_VEL
LIN {X 0,Y 186.76,Z 374.106,A -85,B 0,C 180,E1 -24102.224,E2 -24102.224} C_VEL
LIN {X 0,Y 184.03,Z 370.173,A -85,B 0,C 180,E1 -24104.495,E2 -24104.495} C_VEL
LIN {X 0,Y 181.199,Z 366.085,A -85,B 0,C 180,E1 -24107.185,E2 -24107.185} C_VEL
LIN {X 0,Y 178.624,Z 362.965,A -85,B 0,C 180,E1 -24109.983,E2 -24109.983} C_VEL
LIN {X 0,Y 177.703,Z 361.212,A -85,B 0,C 180,E1 -24111.22,E2 -24111.22} C_VEL
LIN {X 0,Y 174.946,Z 358.26,A -85,B 0,C 180,E1 -24115.391,E2 -24115.391} C_VEL
LIN {X 0,Y 173.955,Z 355.945,A -85,B 0,C 180,E1 -24117.684,E2 -24117.684} C_VEL
LIN {X 0,Y 172.353,Z 355.045,A -85,B 0,C 180,E1 -24122.337,E2 -24122.337} C_VEL
LIN {X 0,Y 171.834,Z 354.795,A -85,B 0,C 180,E1 -24127.048,E2 -24127.048} C_VEL
LIN {X 0,Y 173.794,Z 356.081,A -85,B 0,C 180,E1 -24135.562,E2 -24135.562} C_VEL
LIN {X 0,Y 175.395,Z 359.501,A -85,B 0,C 180,E1 -24139.073,E2 -24139.073} C_VEL
LIN {X 0,Y 177.851,Z 361.895,A -85,B 0,C 180,E1 -24142.585,E2 -24142.585} C_VEL
LIN {X 0,Y 182.276,Z 368.875,A -85,B 0,C 180,E1 -24147.56,E2 -24147.56} C_VEL
LIN {X 0,Y 185.586,Z 374.439,A -85,B 0,C 180,E1 -24150.561,E2 -24150.561} C_VEL
LIN {X 0,Y 188.604,Z 379.889,A -85,B 0,C 180,E1 -24152.977,E2 -24152.977} C_VEL
LIN {X 0,Y 192.717,Z 387.55,A -85,B 0,C 180,E1 -24155.867,E2 -24155.867} C_VEL
LIN {X 0,Y 197.905,Z 398.548,A -85,B 0,C 180,E1 -24159.103,E2 -24159.103} C_VEL
LIN {X 0,Y 202.102,Z 409.111,A -85,B 0,C 180,E1 -24161.52,E2 -24161.52} C_VEL
LIN {X 0,Y 202.349,Z 410.306,A -85,B 0,C 180,E1 -24161.69,E2 -24161.69} C_VEL
LIN {X 0,Y 199.767,Z 440.77,A -85,B 0,C 180,E1 -24162.634,E2 -24162.634} C_VEL
LIN {X 0,Y 197.579,Z 454.175,A -85,B 0,C 180,E1 -24163.351,E2 -24163.351} C_VEL
LIN {X 0,Y 194.563,Z 466.465,A -85,B 0,C 180,E1 -24164.301,E2 -24164.301} C_VEL
LIN {X 0,Y 190.677,Z 478.229,A -85,B 0,C 180,E1 -24165.547,E2 -24165.547} C_VEL
LIN {X 0,Y 186.088,Z 489.561,A -85,B 0,C 180,E1 -24167.17,E2 -24167.17} C_VEL
LIN {X 0,Y 181.254,Z 499.793,A -85,B 0,C 180,E1 -24169.131,E2 -24169.131} C_VEL
LIN {X 0,Y 176.672,Z 508.183,A -85,B 0,C 180,E1 -24171.204,E2 -24171.204} C_VEL
LIN {X 0,Y 170.887,Z 517.315,A -85,B 0,C 180,E1 -24174.121,E2 -24174.121} C_VEL
LIN {X 0,Y 165.667,Z 524.689,A -85,B 0,C 180,E1 -24177.255,E2 -24177.255} C_VEL
LIN {X 0,Y 160.497,Z 531.517,A -85,B 0,C 180,E1 -24181.203,E2 -24181.203} C_VEL
LIN {X 0,Y 156.265,Z 536.479,A -85,B 0,C 180,E1 -24185.187,E2 -24185.187} C_VEL
LIN {X 0,Y 153.46,Z 539.536,A -85,B 0,C 180,E1 -24188.506,E2 -24188.506} C_VEL
LIN {X 0,Y 150.203,Z 542.654,A -85,B 0,C 180,E1 -24193.694,E2 -24193.694} C_VEL
LIN {X 0,Y 149.264,Z 543.536,A -85,B 0,C 180,E1 -24196.107,E2 -24196.107} C_VEL
LIN {X 0,Y 147.961,Z 544.153,A -85,B 0,C 180,E1 -24198.316,E2 -24198.316} C_VEL
LIN {X 0,Y 144.44,Z 544.382,A -85,B 0,C 180,E1 -24201.95,E2 -24201.95} C_VEL
LIN {X 0,Y 141.789,Z 543.921,A -85,B 0,C 180,E1 -24204.966,E2 -24204.966} C_VEL
LIN {X 0,Y 140.735,Z 543.237,A -85,B 0,C 180,E1 -24207.33,E2 -24207.33} C_VEL
LIN {X 0,Y 140.676,Z 542.949,A -85,B 0,C 180,E1 -24208.13,E2 -24208.13} C_VEL
LIN {X 0,Y 140.817,Z 542.242,A -85,B 0,C 180,E1 -24209.998,E2 -24209.998} C_VEL
LIN {X 0,Y 140.657,Z 540.736,A -85,B 0,C 180,E1 -24212.862,E2 -24212.862} C_VEL
LIN {X 0,Y 140.791,Z 537.67,A -85,B 0,C 180,E1 -24217.167,E2 -24217.167} C_VEL
LIN {X 0,Y 141.363,Z 533.509,A -85,B 0,C 180,E1 -24221.468,E2 -24221.468} C_VEL
LIN {X 0,Y 142.755,Z 527.114,A -85,B 0,C 180,E1 -24226.442,E2 -24226.442} C_VEL
LIN {X 0,Y 144.856,Z 520.148,A -85,B 0,C 180,E1 -24230.592,E2 -24230.592} C_VEL
LIN {X 0,Y 146.997,Z 513.052,A -85,B 0,C 180,E1 -24233.95,E2 -24233.95} C_VEL
LIN {X 0,Y 148.358,Z 508.35,A -85,B 0,C 180,E1 -24235.833,E2 -24235.833} C_VEL
LIN {X 0,Y 151.129,Z 499.276,A -85,B 0,C 180,E1 -24238.844,E2 -24238.844} C_VEL
LIN {X 0,Y 154.169,Z 488.609,A -85,B 0,C 180,E1 -24241.615,E2 -24241.615} C_VEL
LIN {X 0,Y 156.811,Z 478.327,A -85,B 0,C 180,E1 -24243.682,E2 -24243.682} C_VEL
LIN {X 0,Y 159.435,Z 466.141,A -85,B 0,C 180,E1 -24245.54,E2 -24245.54} C_VEL
LIN {X 0,Y 161.416,Z 454.063,A -85,B 0,C 180,E1 -24246.869,E2 -24246.869} C_VEL
LIN {X 0,Y 162.905,Z 441.279,A -85,B 0,C 180,E1 -24247.814,E2 -24247.814} C_VEL
LIN {X 0,Y 164.642,Z 412.633,A -85,B 0,C 180,E1 -24249.006,E2 -24249.006} C_VEL
LIN {X 0,Y 165.484,Z 394.945,A -85,B 0,C 180,E1 -24249.729,E2 -24249.729} C_VEL
LIN {X 0,Y 163.961,Z 377.049,A -85,B 0,C 180,E1 -24251.021,E2 -24251.021} C_VEL
LIN {X 0,Y 158.39,Z 361.994,A -85,B 0,C 180,E1 -24253.269,E2 -24253.269} C_VEL
LIN {X 0,Y 153.504,Z 350.975,A -85,B 0,C 180,E1 -24255.308,E2 -24255.308} C_VEL
LIN {X 0,Y 149.661,Z 343.61,A -85,B 0,C 180,E1 -24256.97,E2 -24256.97} C_VEL
LIN {X 0,Y 145.484,Z 337.1,A -85,B 0,C 180,E1 -24258.828,E2 -24258.828} C_VEL
LIN {X 0,Y 143.628,Z 334.645,A -85,B 0,C 180,E1 -24259.678,E2 -24259.678} C_VEL
LIN {X 0,Y 143.08,Z 332.65,A -85,B 0,C 180,E1 -24260.07,E2 -24260.07} C_VEL
LIN {X 0,Y 143.167,Z 332.649,A -85,B 0,C 180,E1 -24266.561,E2 -24266.561} C_VEL
LIN {X 0,Y 143.187,Z 332.645,A -85,B 0,C 180,E1 -24272.06,E2 -24272.06} C_VEL
LIN {X 0,Y 143.271,Z 332.636,A -85,B 0,C 180,E1 -24278.745,E2 -24278.745} C_VEL
LIN {X 0,Y 143.298,Z 332.603,A -85,B 0,C 180,E1 -24282.886,E2 -24282.886} C_VEL
LIN {X 0,Y 143.588,Z 332.598,A -85,B 0,C 180,E1 -24288.71,E2 -24288.71} C_VEL
LIN {X 0,Y 143.659,Z 332.567,A -85,B 0,C 180,E1 -24291.561,E2 -24291.561} C_VEL
LIN {X 0,Y 144.169,Z 332.525,A -85,B 0,C 180,E1 -24300,E2 -24300} C_VEL
LIN {X 0,Y 143.604,Z 332.57,A -85,B 0,C 180,E1 -24308.443,E2 -24308.443} C_VEL
LIN {X 0,Y 143.498,Z 332.608,A -85,B 0,C 180,E1 -24311.628,E2 -24311.628} C_VEL
LIN {X 0,Y 143.289,Z 332.633,A -85,B 0,C 180,E1 -24317.115,E2 -24317.115} C_VEL
LIN {X 0,Y 143.269,Z 332.63,A -85,B 0,C 180,E1 -24321.254,E2 -24321.254} C_VEL
LIN {X 0,Y 143.185,Z 332.638,A -85,B 0,C 180,E1 -24327.938,E2 -24327.938} C_VEL
LIN {X 0,Y 143.141,Z 332.643,A -85,B 0,C 180,E1 -24333.423,E2 -24333.423} C_VEL
LIN {X 0,Y 143.047,Z 332.656,A -85,B 0,C 180,E1 -24339.695,E2 -24339.695} C_VEL
LIN {X 0,Y 143.028,Z 332.66,A -85,B 0,C 180,E1 -24343.466,E2 -24343.466} C_VEL
LIN {X 0,Y 143.033,Z 332.665,A -85,B 0,C 180,E1 -24347.48,E2 -24347.48} C_VEL
LIN {X 0,Y 143.068,Z 332.662,A -85,B 0,C 180,E1 -24351.811,E2 -24351.811} C_VEL
LIN {X 0,Y 143.124,Z 332.786,A -85,B 0,C 180,E1 -24354.609,E2 -24354.609} C_VEL
LIN {X 0,Y 144.018,Z 335.37,A -85,B 0,C 180,E1 -24355.124,E2 -24355.124} C_VEL
LIN {X 0,Y 146.242,Z 338.133,A -85,B 0,C 180,E1 -24356.117,E2 -24356.117} C_VEL
LIN {X 0,Y 148.49,Z 341.469,A -85,B 0,C 180,E1 -24357.111,E2 -24357.111} C_VEL
LIN {X 0,Y 156.012,Z 354.072,A -85,B 0,C 180,E1 -24360.219,E2 -24360.219} C_VEL
LIN {X 0,Y 161.723,Z 365.133,A -85,B 0,C 180,E1 -24362.389,E2 -24362.389} C_VEL
LIN {X 0,Y 166.467,Z 375.586,A -85,B 0,C 180,E1 -24364.103,E2 -24364.103} C_VEL
LIN {X 0,Y 163.26,Z 430.71,A -85,B 0,C 180,E1 -24366.316,E2 -24366.316} C_VEL
LIN {X 0,Y 161.834,Z 444.096,A -85,B 0,C 180,E1 -24367.333,E2 -24367.333} C_VEL
LIN {X 0,Y 159.718,Z 456.598,A -85,B 0,C 180,E1 -24368.716,E2 -24368.716} C_VEL
LIN {X 0,Y 157.542,Z 467.673,A -85,B 0,C 180,E1 -24370.455,E2 -24370.455} C_VEL
LIN {X 0,Y 154.992,Z 478.966,A -85,B 0,C 180,E1 -24372.801,E2 -24372.801} C_VEL
LIN {X 0,Y 151.949,Z 489.64,A -85,B 0,C 180,E1 -24375.606,E2 -24375.606} C_VEL
LIN {X 0,Y 149.362,Z 498.169,A -85,B 0,C 180,E1 -24378.467,E2 -24378.467} C_VEL
LIN {X 0,Y 146.398,Z 507.401,A -85,B 0,C 180,E1 -24382.416,E2 -24382.416} C_VEL
LIN {X 0,Y 144.101,Z 514.821,A -85,B 0,C 180,E1 -24386.507,E2 -24386.507} C_VEL
LIN {X 0,Y 142.699,Z 519.853,A -85,B 0,C 180,E1 -24390.002,E2 -24390.002} C_VEL
LIN {X 0,Y 141.502,Z 524.637,A -85,B 0,C 180,E1 -24394.166,E2 -24394.166} C_VEL
LIN {X 0,Y 140.637,Z 528.53,A -85,B 0,C 180,E1 -24398.624,E2 -24398.624} C_VEL
LIN {X 0,Y 140.337,Z 530.493,A -85,B 0,C 180,E1 -24401.558,E2 -24401.558} C_VEL
LIN {X 0,Y 140.325,Z 531.986,A -85,B 0,C 180,E1 -24404.504,E2 -24404.504} C_VEL
LIN {X 0,Y 140.651,Z 533.291,A -85,B 0,C 180,E1 -24408.306,E2 -24408.306} C_VEL
LIN {X 0,Y 141.671,Z 533.968,A -85,B 0,C 180,E1 -24413.384,E2 -24413.384} C_VEL
LIN {X 0,Y 143.582,Z 533.417,A -85,B 0,C 180,E1 -24418.229,E2 -24418.229} C_VEL
LIN {X 0,Y 145.675,Z 532.131,A -85,B 0,C 180,E1 -24422.054,E2 -24422.054} C_VEL
LIN {X 0,Y 149.259,Z 529.269,A -85,B 0,C 180,E1 -24426.825,E2 -24426.825} C_VEL
LIN {X 0,Y 153.824,Z 524.836,A -85,B 0,C 180,E1 -24431.491,E2 -24431.491} C_VEL
LIN {X 0,Y 158.441,Z 519.776,A -85,B 0,C 180,E1 -24435.213,E2 -24435.213} C_VEL
LIN {X 0,Y 163.633,Z 513.332,A -85,B 0,C 180,E1 -24438.733,E2 -24438.733} C_VEL
LIN {X 0,Y 169.463,Z 505.159,A -85,B 0,C 180,E1 -24441.998,E2 -24441.998} C_VEL
LIN {X 0,Y 174.683,Z 496.746,A -85,B 0,C 180,E1 -24444.561,E2 -24444.561} C_VEL
LIN {X 0,Y 180.114,Z 486.716,A -85,B 0,C 180,E1 -24446.888,E2 -24446.888} C_VEL
LIN {X 0,Y 184.861,Z 475.984,A -85,B 0,C 180,E1 -24448.805,E2 -24448.805} C_VEL
LIN {X 0,Y 189.018,Z 464.539,A -85,B 0,C 180,E1 -24450.358,E2 -24450.358} C_VEL
LIN {X 0,Y 192.524,Z 452.254,A -85,B 0,C 180,E1 -24451.597,E2 -24451.597} C_VEL
LIN {X 0,Y 195.136,Z 439.267,A -85,B 0,C 180,E1 -24452.518,E2 -24452.518} C_VEL
LIN {X 0,Y 196.857,Z 425.863,A -85,B 0,C 180,E1 -24453.104,E2 -24453.104} C_VEL
LIN {X 0,Y 198.635,Z 404.429,A -85,B 0,C 180,E1 -24453.734,E2 -24453.734} C_VEL
LIN {X 0,Y 195.085,Z 397.495,A -85,B 0,C 180,E1 -24455.791,E2 -24455.791} C_VEL
LIN {X 0,Y 190.831,Z 390.056,A -85,B 0,C 180,E1 -24458.47,E2 -24458.47} C_VEL
LIN {X 0,Y 186.794,Z 383.59,A -85,B 0,C 180,E1 -24461.361,E2 -24461.361} C_VEL
LIN {X 0,Y 184.325,Z 379.867,A -85,B 0,C 180,E1 -24463.336,E2 -24463.336} C_VEL
LIN {X 0,Y 182.117,Z 376.535,A -85,B 0,C 180,E1 -24465.294,E2 -24465.294} C_VEL
LIN {X 0,Y 179.462,Z 372.635,A -85,B 0,C 180,E1 -24467.956,E2 -24467.956} C_VEL
LIN {X 0,Y 176.803,Z 368.985,A -85,B 0,C 180,E1 -24471.097,E2 -24471.097} C_VEL
LIN {X 0,Y 176.128,Z 367.864,A -85,B 0,C 180,E1 -24472.051,E2 -24472.051} C_VEL
LIN {X 0,Y 173.624,Z 364.787,A -85,B 0,C 180,E1 -24476.215,E2 -24476.215} C_VEL
LIN {X 0,Y 172.786,Z 362.855,A -85,B 0,C 180,E1 -24478.309,E2 -24478.309} C_VEL
LIN {X 0,Y 171.47,Z 362.092,A -85,B 0,C 180,E1 -24482.349,E2 -24482.349} C_VEL
LIN {X 0,Y 170.958,Z 361.845,A -85,B 0,C 180,E1 -24487.084,E2 -24487.084} C_VEL
LIN {X 0,Y 172.768,Z 363.148,A -85,B 0,C 180,E1 -24495.273,E2 -24495.273} C_VEL
LIN {X 0,Y 174.205,Z 366.353,A -85,B 0,C 180,E1 -24498.605,E2 -24498.605} C_VEL
LIN {X 0,Y 176.556,Z 368.736,A -85,B 0,C 180,E1 -24502.126,E2 -24502.126} C_VEL
LIN {X 0,Y 180.523,Z 375.382,A -85,B 0,C 180,E1 -24506.827,E2 -24506.827} C_VEL
LIN {X 0,Y 183.468,Z 380.577,A -85,B 0,C 180,E1 -24509.663,E2 -24509.663} C_VEL
LIN {X 0,Y 186.373,Z 386.092,A -85,B 0,C 180,E1 -24512.132,E2 -24512.132} C_VEL
LIN {X 0,Y 190.232,Z 393.727,A -85,B 0,C 180,E1 -24515.025,E2 -24515.025} C_VEL
LIN {X 0,Y 194.767,Z 403.802,A -85,B 0,C 180,E1 -24518.031,E2 -24518.031} C_VEL
LIN {X 0,Y 198.061,Z 412.402,A -85,B 0,C 180,E1 -24520.07,E2 -24520.07} C_VEL
LIN {X 0,Y 195.722,Z 439.738,A -85,B 0,C 180,E1 -24520.928,E2 -24520.928} C_VEL
LIN {X 0,Y 193.431,Z 453.539,A -85,B 0,C 180,E1 -24521.65,E2 -24521.65} C_VEL
LIN {X 0,Y 190.326,Z 465.908,A -85,B 0,C 180,E1 -24522.589,E2 -24522.589} C_VEL
LIN {X 0,Y 186.314,Z 477.742,A -85,B 0,C 180,E1 -24523.827,E2 -24523.827} C_VEL
LIN {X 0,Y 181.573,Z 489.112,A -85,B 0,C 180,E1 -24525.447,E2 -24525.447} C_VEL
LIN {X 0,Y 176.519,Z 499.38,A -85,B 0,C 180,E1 -24527.401,E2 -24527.401} C_VEL
LIN {X 0,Y 171.211,Z 508.635,A -85,B 0,C 180,E1 -24529.719,E2 -24529.719} C_VEL
LIN {X 0,Y 165.202,Z 517.63,A -85,B 0,C 180,E1 -24532.682,E2 -24532.682} C_VEL
LIN {X 0,Y 159.75,Z 524.903,A -85,B 0,C 180,E1 -24535.879,E2 -24535.879} C_VEL
LIN {X 0,Y 155.762,Z 529.848,A -85,B 0,C 180,E1 -24538.741,E2 -24538.741} C_VEL
LIN {X 0,Y 151.574,Z 534.681,A -85,B 0,C 180,E1 -24542.374,E2 -24542.374} C_VEL
LIN {X 0,Y 147.905,Z 538.426,A -85,B 0,C 180,E1 -24546.176,E2 -24546.176} C_VEL
LIN {X 0,Y 144.939,Z 541.184,A -85,B 0,C 180,E1 -24550.156,E2 -24550.156} C_VEL
LIN {X 0,Y 142.253,Z 543.45,A -85,B 0,C 180,E1 -24555.697,E2 -24555.697} C_VEL
LIN {X 0,Y 141.426,Z 543.996,A -85,B 0,C 180,E1 -24558.533,E2 -24558.533} C_VEL
LIN {X 0,Y 140.683,Z 543.888,A -85,B 0,C 180,E1 -24564.264,E2 -24564.264} C_VEL
LIN {X 0,Y 140.676,Z 542.949,A -85,B 0,C 180,E1 -24568.13,E2 -24568.13} C_VEL
LIN {X 0,Y 140.046,Z 541.966,A -85,B 0,C 180,E1 -24570.48,E2 -24570.48} C_VEL
LIN {X 0,Y 138.462,Z 540.684,A -85,B 0,C 180,E1 -24572.777,E2 -24572.777} C_VEL
LIN {X 0,Y 134.855,Z 537.309,A -85,B 0,C 180,E1 -24577.39,E2 -24577.39} C_VEL
LIN {X 0,Y 134.053,Z 535.217,A -85,B 0,C 180,E1 -24579.769,E2 -24579.769} C_VEL
LIN {X 0,Y 134.094,Z 534.451,A -85,B 0,C 180,E1 -24580.565,E2 -24580.565} C_VEL
LIN {X 0,Y 135.119,Z 529.417,A -85,B 0,C 180,E1 -24585.072,E2 -24585.072} C_VEL
LIN {X 0,Y 137.017,Z 523.089,A -85,B 0,C 180,E1 -24589.473,E2 -24589.473} C_VEL
LIN {X 0,Y 139.564,Z 515.126,A -85,B 0,C 180,E1 -24593.754,E2 -24593.754} C_VEL
LIN {X 0,Y 141.606,Z 508.366,A -85,B 0,C 180,E1 -24596.702,E2 -24596.702} C_VEL
LIN {X 0,Y 144.571,Z 499.18,A -85,B 0,C 180,E1 -24599.884,E2 -24599.884} C_VEL
LIN {X 0,Y 147.751,Z 488.545,A -85,B 0,C 180,E1 -24602.754,E2 -24602.754} C_VEL
LIN {X 0,Y 150.507,Z 478.304,A -85,B 0,C 180,E1 -24604.888,E2 -24604.888} C_VEL
LIN {X 0,Y 153.239,Z 466.213,A -85,B 0,C 180,E1 -24606.802,E2 -24606.802} C_VEL
LIN {X 0,Y 155.301,Z 454.247,A -85,B 0,C 180,E1 -24608.167,E2 -24608.167} C_VEL
LIN {X 0,Y 156.872,Z 441.587,A -85,B 0,C 180,E1 -24609.139,E2 -24609.139} C_VEL
LIN {X 0,Y 158.362,Z 418.96,A -85,B 0,C 180,E1 -24610.129,E2 -24610.129} C_VEL
LIN {X 0,Y 159.527,Z 395.361,A -85,B 0,C 180,E1 -24611.125,E2 -24611.125} C_VEL
LIN {X 0,Y 158.269,Z 379.495,A -85,B 0,C 180,E1 -24612.321,E2 -24612.321} C_VEL
LIN {X 0,Y 153.216,Z 365.48,A -85,B 0,C 180,E1 -24614.529,E2 -24614.529} C_VEL
LIN {X 0,Y 148.169,Z 353.892,A -85,B 0,C 180,E1 -24616.809,E2 -24616.809} C_VEL
LIN {X 0,Y 145.108,Z 348.027,A -85,B 0,C 180,E1 -24618.235,E2 -24618.235} C_VEL
LIN {X 0,Y 141.227,Z 342.093,A -85,B 0,C 180,E1 -24620.076,E2 -24620.076} C_VEL
LIN {X 0,Y 138.474,Z 338.013,A -85,B 0,C 180,E1 -24621.47,E2 -24621.47} C_VEL
LIN {X 0,Y 136.713,Z 335.766,A -85,B 0,C 180,E1 -24622.377,E2 -24622.377} C_VEL
LIN {X 0,Y 136.042,Z 333.539,A -85,B 0,C 180,E1 -24622.859,E2 -24622.859} C_VEL
LIN {X 0,Y 136.087,Z 333.532,A -85,B 0,C 180,E1 -24625.715,E2 -24625.715} C_VEL
LIN {X 0,Y 136.143,Z 333.523,A -85,B 0,C 180,E1 -24632.316,E2 -24632.316} C_VEL
LIN {X 0,Y 136.238,Z 333.511,A -85,B 0,C 180,E1 -24638.832,E2 -24638.832} C_VEL
LIN {X 0,Y 136.269,Z 333.49,A -85,B 0,C 180,E1 -24645.056,E2 -24645.056} C_VEL
LIN {X 0,Y 136.491,Z 333.482,A -85,B 0,C 180,E1 -24648.114,E2 -24648.114} C_VEL
LIN {X 0,Y 136.586,Z 333.452,A -85,B 0,C 180,E1 -24651.12,E2 -24651.12} C_VEL
LIN {X 0,Y 137.126,Z 333.402,A -85,B 0,C 180,E1 -24660,E2 -24660} C_VEL
LIN {X 0,Y 136.533,Z 333.453,A -85,B 0,C 180,E1 -24668.884,E2 -24668.884} C_VEL
LIN {X 0,Y 136.435,Z 333.489,A -85,B 0,C 180,E1 -24671.891,E2 -24671.891} C_VEL
LIN {X 0,Y 136.232,Z 333.514,A -85,B 0,C 180,E1 -24678.031,E2 -24678.031} C_VEL
LIN {X 0,Y 136.191,Z 333.51,A -85,B 0,C 180,E1 -24681.748,E2 -24681.748} C_VEL
LIN {X 0,Y 136.111,Z 333.52,A -85,B 0,C 180,E1 -24688.63,E2 -24688.63} C_VEL
LIN {X 0,Y 136.038,Z 333.529,A -85,B 0,C 180,E1 -24694.631,E2 -24694.631} C_VEL
LIN {X 0,Y 136.019,Z 333.531,A -85,B 0,C 180,E1 -24699.196,E2 -24699.196} C_VEL
LIN {X 0,Y 135.973,Z 333.538,A -85,B 0,C 180,E1 -24703.65,E2 -24703.65} C_VEL
LIN {X 0,Y 135.978,Z 333.542,A -85,B 0,C 180,E1 -24707.789,E2 -24707.789} C_VEL
LIN {X 0,Y 136.02,Z 333.541,A -85,B 0,C 180,E1 -24711.75,E2 -24711.75} C_VEL
LIN {X 0,Y 136.953,Z 336.255,A -85,B 0,C 180,E1 -24712.361,E2 -24712.361} C_VEL
LIN {X 0,Y 139.312,Z 339.116,A -85,B 0,C 180,E1 -24713.556,E2 -24713.556} C_VEL
LIN {X 0,Y 141.615,Z 342.498,A -85,B 0,C 180,E1 -24714.707,E2 -24714.707} C_VEL
LIN {X 0,Y 147.28,Z 351.405,A -85,B 0,C 180,E1 -24717.341,E2 -24717.341} C_VEL
LIN {X 0,Y 154.098,Z 363.635,A -85,B 0,C 180,E1 -24720.225,E2 -24720.225} C_VEL
LIN {X 0,Y 160.534,Z 377.539,A -85,B 0,C 180,E1 -24722.762,E2 -24722.762} C_VEL
LIN {X 0,Y 157.305,Z 430.639,A -85,B 0,C 180,E1 -24724.941,E2 -24724.941} C_VEL
LIN {X 0,Y 155.803,Z 444.259,A -85,B 0,C 180,E1 -24725.998,E2 -24725.998} C_VEL
LIN {X 0,Y 153.724,Z 456.018,A -85,B 0,C 180,E1 -24727.312,E2 -24727.312} C_VEL
LIN {X 0,Y 151.247,Z 468.122,A -85,B 0,C 180,E1 -24729.251,E2 -24729.251} C_VEL
LIN {X 0,Y 148.404,Z 480.011,A -85,B 0,C 180,E1 -24731.83,E2 -24731.83} C_VEL
LIN {X 0,Y 145.187,Z 490.75,A -85,B 0,C 180,E1 -24734.814,E2 -24734.814} C_VEL
LIN {X 0,Y 141.834,Z 501.013,A -85,B 0,C 180,E1 -24738.57,E2 -24738.57} C_VEL
LIN {X 0,Y 138.926,Z 509.776,A -85,B 0,C 180,E1 -24742.737,E2 -24742.737} C_VEL
LIN {X 0,Y 136.665,Z 516.76,A -85,B 0,C 180,E1 -24747.054,E2 -24747.054} C_VEL
LIN {X 0,Y 135.038,Z 522.355,A -85,B 0,C 180,E1 -24751.493,E2 -24751.493} C_VEL
LIN {X 0,Y 133.951,Z 526.759,A -85,B 0,C 180,E1 -24756.025,E2 -24756.025} C_VEL
LIN {X 0,Y 133.469,Z 529.104,A -85,B 0,C 180,E1 -24759.091,E2 -24759.091} C_VEL
LIN {X 0,Y 133.205,Z 531,A -85,B 0,C 180,E1 -24762.186,E2 -24762.186} C_VEL
LIN {X 0,Y 133.277,Z 532.418,A -85,B 0,C 180,E1 -24765.29,E2 -24765.29} C_VEL
LIN {X 0,Y 133.593,Z 533.529,A -85,B 0,C 180,E1 -24768.748,E2 -24768.748} C_VEL
LIN {X 0,Y 134.067,Z 534.056,A -85,B 0,C 180,E1 -24771.53,E2 -24771.53} C_VEL
LIN {X 0,Y 134.911,Z 534.223,A -85,B 0,C 180,E1 -24774.631,E2 -24774.631} C_VEL
LIN {X 0,Y 136.792,Z 533.722,A -85,B 0,C 180,E1 -24779.141,E2 -24779.141} C_VEL
LIN {X 0,Y 139.433,Z 532.22,A -85,B 0,C 180,E1 -24783.674,E2 -24783.674} C_VEL
LIN {X 0,Y 142.896,Z 529.63,A -85,B 0,C 180,E1 -24788.101,E2 -24788.101} C_VEL
LIN {X 0,Y 146.83,Z 526.153,A -85,B 0,C 180,E1 -24792.077,E2 -24792.077} C_VEL
LIN {X 0,Y 151.561,Z 521.406,A -85,B 0,C 180,E1 -24795.928,E2 -24795.928} C_VEL
LIN {X 0,Y 156.91,Z 515.259,A -85,B 0,C 180,E1 -24799.593,E2 -24799.593} C_VEL
LIN {X 0,Y 162.55,Z 508.074,A -85,B 0,C 180,E1 -24802.749,E2 -24802.749} C_VEL
LIN {X 0,Y 168.272,Z 499.644,A -85,B 0,C 180,E1 -24805.577,E2 -24805.577} C_VEL
LIN {X 0,Y 173.996,Z 489.872,A -85,B 0,C 180,E1 -24808.021,E2 -24808.021} C_VEL
LIN {X 0,Y 179.31,Z 478.899,A -85,B 0,C 180,E1 -24810.135,E2 -24810.135} C_VEL
LIN {X 0,Y 183.606,Z 468.216,A -85,B 0,C 180,E1 -24811.691,E2 -24811.691} C_VEL
LIN {X 0,Y 187.372,Z 456.404,A -85,B 0,C 180,E1 -24812.978,E2 -24812.978} C_VEL
LIN {X 0,Y 190.512,Z 442.89,A -85,B 0,C 180,E1 -24814.048,E2 -24814.048} C_VEL
LIN {X 0,Y 192.407,Z 430.851,A -85,B 0,C 180,E1 -24814.665,E2 -24814.665} C_VEL
LIN {X 0,Y 194.46,Z 407.393,A -85,B 0,C 180,E1 -24815.4,E2 -24815.4} C_VEL
LIN {X 0,Y 189.42,Z 397.751,A -85,B 0,C 180,E1 -24818.642,E2 -24818.642} C_VEL
LIN {X 0,Y 184.827,Z 390.085,A -85,B 0,C 180,E1 -24822.048,E2 -24822.048} C_VEL
LIN {X 0,Y 181.727,Z 385.201,A -85,B 0,C 180,E1 -24824.697,E2 -24824.697} C_VEL
LIN {X 0,Y 180.016,Z 382.61,A -85,B 0,C 180,E1 -24826.327,E2 -24826.327} C_VEL
LIN {X 0,Y 177.741,Z 379.117,A -85,B 0,C 180,E1 -24828.764,E2 -24828.764} C_VEL
LIN {X 0,Y 175.2,Z 375.309,A -85,B 0,C 180,E1 -24832.008,E2 -24832.008} C_VEL
LIN {X 0,Y 174.286,Z 374.157,A -85,B 0,C 180,E1 -24833.379,E2 -24833.379} C_VEL
LIN {X 0,Y 172.285,Z 371.191,A -85,B 0,C 180,E1 -24837.183,E2 -24837.183} C_VEL
LIN {X 0,Y 171.77,Z 369.815,A -85,B 0,C 180,E1 -24838.62,E2 -24838.62} C_VEL
LIN {X 0,Y 170.59,Z 369.12,A -85,B 0,C 180,E1 -24842.361,E2 -24842.361} C_VEL
LIN {X 0,Y 170.271,Z 369.075,A -85,B 0,C 180,E1 -24849.503,E2 -24849.503} C_VEL
LIN {X 0,Y 171.707,Z 370.21,A -85,B 0,C 180,E1 -24854.888,E2 -24854.888} C_VEL
LIN {X 0,Y 173.228,Z 373.443,A -85,B 0,C 180,E1 -24858.488,E2 -24858.488} C_VEL
LIN {X 0,Y 175.207,Z 375.556,A -85,B 0,C 180,E1 -24861.577,E2 -24861.577} C_VEL
LIN {X 0,Y 178.788,Z 381.893,A -85,B 0,C 180,E1 -24866.075,E2 -24866.075} C_VEL
LIN {X 0,Y 181.515,Z 386.958,A -85,B 0,C 180,E1 -24868.859,E2 -24868.859} C_VEL
LIN {X 0,Y 184.483,Z 392.877,A -85,B 0,C 180,E1 -24871.518,E2 -24871.518} C_VEL
LIN {X 0,Y 188.527,Z 401.421,A -85,B 0,C 180,E1 -24874.692,E2 -24874.692} C_VEL
LIN {X 0,Y 192.482,Z 411.029,A -85,B 0,C 180,E1 -24877.45,E2 -24877.45} C_VEL
LIN {X 0,Y 193.963,Z 415.087,A -85,B 0,C 180,E1 -24878.432,E2 -24878.432} C_VEL
LIN {X 0,Y 191.645,Z 440.216,A -85,B 0,C 180,E1 -24879.215,E2 -24879.215} C_VEL
LIN {X 0,Y 189.312,Z 453.62,A -85,B 0,C 180,E1 -24879.921,E2 -24879.921} C_VEL
LIN {X 0,Y 185.946,Z 466.372,A -85,B 0,C 180,E1 -24880.893,E2 -24880.893} C_VEL
LIN {X 0,Y 181.499,Z 478.827,A -85,B 0,C 180,E1 -24882.22,E2 -24882.22} C_VEL
LIN {X 0,Y 176.617,Z 489.95,A -85,B 0,C 180,E1 -24883.842,E2 -24883.842} C_VEL
LIN {X 0,Y 171.379,Z 499.987,A -85,B 0,C 180,E1 -24885.8,E2 -24885.8} C_VEL
LIN {X 0,Y 165.88,Z 509.066,A -85,B 0,C 180,E1 -24888.14,E2 -24888.14} C_VEL
LIN {X 0,Y 160.639,Z 516.594,A -85,B 0,C 180,E1 -24890.624,E2 -24890.624} C_VEL
LIN {X 0,Y 154.839,Z 524,A -85,B 0,C 180,E1 -24893.837,E2 -24893.837} C_VEL
LIN {X 0,Y 149.738,Z 529.971,A -85,B 0,C 180,E1 -24897.331,E2 -24897.331} C_VEL
LIN {X 0,Y 145.304,Z 534.721,A -85,B 0,C 180,E1 -24901.072,E2 -24901.072} C_VEL
LIN {X 0,Y 141.406,Z 538.388,A -85,B 0,C 180,E1 -24905.008,E2 -24905.008} C_VEL
LIN {X 0,Y 138.254,Z 541.073,A -85,B 0,C 180,E1 -24909.153,E2 -24909.153} C_VEL
LIN {X 0,Y 136.566,Z 542.361,A -85,B 0,C 180,E1 -24912.013,E2 -24912.013} C_VEL
LIN {X 0,Y 135.36,Z 543.265,A -85,B 0,C 180,E1 -24914.951,E2 -24914.951} C_VEL
LIN {X 0,Y 133.866,Z 543.847,A -85,B 0,C 180,E1 -24920.936,E2 -24920.936} C_VEL
LIN {X 0,Y 133.616,Z 543.572,A -85,B 0,C 180,E1 -24923.959,E2 -24923.959} C_VEL
LIN {X 0,Y 133.612,Z 542.536,A -85,B 0,C 180,E1 -24928.125,E2 -24928.125} C_VEL
LIN {X 0,Y 133.718,Z 541.833,A -85,B 0,C 180,E1 -24929.998,E2 -24929.998} C_VEL
LIN {X 0,Y 133.569,Z 540.285,A -85,B 0,C 180,E1 -24933.014,E2 -24933.014} C_VEL
LIN {X 0,Y 133.748,Z 537.146,A -85,B 0,C 180,E1 -24937.546,E2 -24937.546} C_VEL
LIN {X 0,Y 134.094,Z 534.451,A -85,B 0,C 180,E1 -24940.565,E2 -24940.565} C_VEL
LIN {X 0,Y 133.924,Z 532.093,A -85,B 0,C 180,E1 -24942.877,E2 -24942.877} C_VEL
LIN {X 0,Y 132.244,Z 527.679,A -85,B 0,C 180,E1 -24946.627,E2 -24946.627} C_VEL
LIN {X 0,Y 130.912,Z 522.581,A -85,B 0,C 180,E1 -24950.305,E2 -24950.305} C_VEL
LIN {X 0,Y 131.289,Z 519.147,A -85,B 0,C 180,E1 -24952.414,E2 -24952.414} C_VEL
LIN {X 0,Y 133.633,Z 512.063,A -85,B 0,C 180,E1 -24956.048,E2 -24956.048} C_VEL
LIN {X 0,Y 136.492,Z 504.114,A -85,B 0,C 180,E1 -24959.282,E2 -24959.282} C_VEL
LIN {X 0,Y 139.437,Z 494.633,A -85,B 0,C 180,E1 -24962.377,E2 -24962.377} C_VEL
LIN {X 0,Y 142.604,Z 484.354,A -85,B 0,C 180,E1 -24964.951,E2 -24964.951} C_VEL
LIN {X 0,Y 145.54,Z 473.094,A -85,B 0,C 180,E1 -24967.126,E2 -24967.126} C_VEL
LIN {X 0,Y 147.946,Z 461.677,A -85,B 0,C 180,E1 -24968.786,E2 -24968.786} C_VEL
LIN {X 0,Y 150.156,Z 448.85,A -85,B 0,C 180,E1 -24970.055,E2 -24970.055} C_VEL
LIN {X 0,Y 151.468,Z 435.777,A -85,B 0,C 180,E1 -24970.9,E2 -24970.9} C_VEL
LIN {X 0,Y 153.722,Z 395.904,A -85,B 0,C 180,E1 -24972.608,E2 -24972.608} C_VEL
LIN {X 0,Y 152.61,Z 381.617,A -85,B 0,C 180,E1 -24973.751,E2 -24973.751} C_VEL
LIN {X 0,Y 147.932,Z 368.425,A -85,B 0,C 180,E1 -24975.969,E2 -24975.969} C_VEL
LIN {X 0,Y 143.15,Z 357.297,A -85,B 0,C 180,E1 -24978.313,E2 -24978.313} C_VEL
LIN {X 0,Y 139.945,Z 351.243,A -85,B 0,C 180,E1 -24979.929,E2 -24979.929} C_VEL
LIN {X 0,Y 136.768,Z 346.544,A -85,B 0,C 180,E1 -24981.556,E2 -24981.556} C_VEL
LIN {X 0,Y 134.584,Z 343.303,A -85,B 0,C 180,E1 -24982.74,E2 -24982.74} C_VEL
LIN {X 0,Y 132.479,Z 340.119,A -85,B 0,C 180,E1 -24983.948,E2 -24983.948} C_VEL
LIN {X 0,Y 131.69,Z 339.135,A -85,B 0,C 180,E1 -24984.401,E2 -24984.401} C_VEL
LIN {X 0,Y 129.78,Z 336.789,A -85,B 0,C 180,E1 -24985.534,E2 -24985.534} C_VEL
LIN {X 0,Y 129.015,Z 334.413,A -85,B 0,C 180,E1 -24986.151,E2 -24986.151} C_VEL
LIN {X 0,Y 129.046,Z 334.405,A -85,B 0,C 180,E1 -24990.65,E2 -24990.65} C_VEL
LIN {X 0,Y 129.102,Z 334.404,A -85,B 0,C 180,E1 -24997.727,E2 -24997.727} C_VEL
LIN {X 0,Y 129.148,Z 334.372,A -85,B 0,C 180,E1 -25000.943,E2 -25000.943} C_VEL
LIN {X 0,Y 129.41,Z 334.365,A -85,B 0,C 180,E1 -25007.82,E2 -25007.82} C_VEL
LIN {X 0,Y 129.511,Z 334.337,A -85,B 0,C 180,E1 -25010.631,E2 -25010.631} C_VEL
LIN {X 0,Y 130.08,Z 334.28,A -85,B 0,C 180,E1 -25020,E2 -25020} C_VEL
LIN {X 0,Y 129.459,Z 334.338,A -85,B 0,C 180,E1 -25029.373,E2 -25029.373} C_VEL
LIN {X 0,Y 129.338,Z 334.373,A -85,B 0,C 180,E1 -25032.554,E2 -25032.554} C_VEL
LIN {X 0,Y 129.145,Z 334.398,A -85,B 0,C 180,E1 -25039.058,E2 -25039.058} C_VEL
LIN {X 0,Y 129.102,Z 334.393,A -85,B 0,C 180,E1 -25042.4,E2 -25042.4} C_VEL
LIN {X 0,Y 129.031,Z 334.405,A -85,B 0,C 180,E1 -25049.375,E2 -25049.375} C_VEL
LIN {X 0,Y 128.954,Z 334.414,A -85,B 0,C 180,E1 -25055.169,E2 -25055.169} C_VEL
LIN {X 0,Y 128.918,Z 334.421,A -85,B 0,C 180,E1 -25060.858,E2 -25060.858} C_VEL
LIN {X 0,Y 128.923,Z 334.423,A -85,B 0,C 180,E1 -25067.386,E2 -25067.386} C_VEL
LIN {X 0,Y 128.934,Z 334.417,A -85,B 0,C 180,E1 -25068.391,E2 -25068.391} C_VEL
LIN {X 0,Y 129.871,Z 337.184,A -85,B 0,C 180,E1 -25069.147,E2 -25069.147} C_VEL
LIN {X 0,Y 132.006,Z 339.391,A -85,B 0,C 180,E1 -25070.371,E2 -25070.371} C_VEL
LIN {X 0,Y 134.514,Z 343.268,A -85,B 0,C 180,E1 -25071.826,E2 -25071.826} C_VEL
LIN {X 0,Y 136.22,Z 345.73,A -85,B 0,C 180,E1 -25072.753,E2 -25072.753} C_VEL
LIN {X 0,Y 140.546,Z 352.125,A -85,B 0,C 180,E1 -25074.969,E2 -25074.969} C_VEL
LIN {X 0,Y 147.63,Z 364.512,A -85,B 0,C 180,E1 -25078.291,E2 -25078.291} C_VEL
LIN {X 0,Y 153.836,Z 377.7,A -85,B 0,C 180,E1 -25080.973,E2 -25080.973} C_VEL
LIN {X 0,Y 154.719,Z 380.097,A -85,B 0,C 180,E1 -25081.36,E2 -25081.36} C_VEL
LIN {X 0,Y 151.372,Z 431.294,A -85,B 0,C 180,E1 -25083.503,E2 -25083.503} C_VEL
LIN {X 0,Y 149.74,Z 445.19,A -85,B 0,C 180,E1 -25084.627,E2 -25084.627} C_VEL
LIN {X 0,Y 147.405,Z 457.606,A -85,B 0,C 180,E1 -25086.095,E2 -25086.095} C_VEL
LIN {X 0,Y 144.654,Z 470.147,A -85,B 0,C 180,E1 -25088.259,E2 -25088.259} C_VEL
LIN {X 0,Y 141.879,Z 480.992,A -85,B 0,C 180,E1 -25090.752,E2 -25090.752} C_VEL
LIN {X 0,Y 138.559,Z 491.423,A -85,B 0,C 180,E1 -25093.804,E2 -25093.804} C_VEL
LIN {X 0,Y 135.44,Z 500.549,A -85,B 0,C 180,E1 -25097.262,E2 -25097.262} C_VEL
LIN {X 0,Y 132.32,Z 509.446,A -85,B 0,C 180,E1 -25101.604,E2 -25101.604} C_VEL
LIN {X 0,Y 129.855,Z 516.575,A -85,B 0,C 180,E1 -25106.123,E2 -25106.123} C_VEL
LIN {X 0,Y 128.354,Z 521.409,A -85,B 0,C 180,E1 -25110.002,E2 -25110.002} C_VEL
LIN {X 0,Y 127.019,Z 526.42,A -85,B 0,C 180,E1 -25115.155,E2 -25115.155} C_VEL
LIN {X 0,Y 126.298,Z 529.677,A -85,B 0,C 180,E1 -25119.612,E2 -25119.612} C_VEL
LIN {X 0,Y 126.089,Z 531.48,A -85,B 0,C 180,E1 -25122.885,E2 -25122.885} C_VEL
LIN {X 0,Y 126.22,Z 532.852,A -85,B 0,C 180,E1 -25126.167,E2 -25126.167} C_VEL
LIN {X 0,Y 126.574,Z 533.826,A -85,B 0,C 180,E1 -25129.462,E2 -25129.462} C_VEL
LIN {X 0,Y 127.234,Z 534.371,A -85,B 0,C 180,E1 -25132.749,E2 -25132.749} C_VEL
LIN {X 0,Y 128.227,Z 534.473,A -85,B 0,C 180,E1 -25136.009,E2 -25136.009} C_VEL
LIN {X 0,Y 130.05,Z 534.022,A -85,B 0,C 180,E1 -25140.156,E2 -25140.156} C_VEL
LIN {X 0,Y 133.298,Z 532.283,A -85,B 0,C 180,E1 -25145.45,E2 -25145.45} C_VEL
LIN {X 0,Y 136.655,Z 529.969,A -85,B 0,C 180,E1 -25149.517,E2 -25149.517} C_VEL
LIN {X 0,Y 141.39,Z 526.011,A -85,B 0,C 180,E1 -25154.1,E2 -25154.1} C_VEL
LIN {X 0,Y 146.709,Z 520.911,A -85,B 0,C 180,E1 -25158.186,E2 -25158.186} C_VEL
LIN {X 0,Y 152.192,Z 514.88,A -85,B 0,C 180,E1 -25161.726,E2 -25161.726} C_VEL
LIN {X 0,Y 157.435,Z 508.491,A -85,B 0,C 180,E1 -25164.526,E2 -25164.526} C_VEL
LIN {X 0,Y 163.044,Z 500.651,A -85,B 0,C 180,E1 -25167.2,E2 -25167.2} C_VEL
LIN {X 0,Y 168.975,Z 491.109,A -85,B 0,C 180,E1 -25169.661,E2 -25169.661} C_VEL
LIN {X 0,Y 174.436,Z 480.456,A -85,B 0,C 180,E1 -25171.755,E2 -25171.755} C_VEL
LIN {X 0,Y 178.916,Z 469.922,A -85,B 0,C 180,E1 -25173.337,E2 -25173.337} C_VEL
LIN {X 0,Y 183.08,Z 457.793,A -85,B 0,C 180,E1 -25174.693,E2 -25174.693} C_VEL
LIN {X 0,Y 186.282,Z 444.969,A -85,B 0,C 180,E1 -25175.729,E2 -25175.729} C_VEL
LIN {X 0,Y 188.421,Z 432.561,A -85,B 0,C 180,E1 -25176.394,E2 -25176.394} C_VEL
LIN {X 0,Y 190.481,Z 410.665,A -85,B 0,C 180,E1 -25177.104,E2 -25177.104} C_VEL
LIN {X 0,Y 186.032,Z 402.097,A -85,B 0,C 180,E1 -25180.242,E2 -25180.242} C_VEL
LIN {X 0,Y 182.057,Z 395.219,A -85,B 0,C 180,E1 -25183.459,E2 -25183.459} C_VEL
LIN {X 0,Y 178.79,Z 389.737,A -85,B 0,C 180,E1 -25186.557,E2 -25186.557} C_VEL
LIN {X 0,Y 175.994,Z 385.514,A -85,B 0,C 180,E1 -25189.664,E2 -25189.664} C_VEL
LIN {X 0,Y 173.392,Z 381.317,A -85,B 0,C 180,E1 -25193.344,E2 -25193.344} C_VEL
LIN {X 0,Y 171.222,Z 378.213,A -85,B 0,C 180,E1 -25197.527,E2 -25197.527} C_VEL
LIN {X 0,Y 170.754,Z 376.804,A -85,B 0,C 180,E1 -25198.936,E2 -25198.936} C_VEL
LIN {X 0,Y 169.289,Z 376.041,A -85,B 0,C 180,E1 -25204.883,E2 -25204.883} C_VEL
LIN {X 0,Y 169.397,Z 376.143,A -85,B 0,C 180,E1 -25209.553,E2 -25209.553} C_VEL
LIN {X 0,Y 170.657,Z 377.234,A -85,B 0,C 180,E1 -25214.499,E2 -25214.499} C_VEL
LIN {X 0,Y 172.253,Z 380.512,A -85,B 0,C 180,E1 -25218.37,E2 -25218.37} C_VEL
LIN {X 0,Y 173.852,Z 382.341,A -85,B 0,C 180,E1 -25220.982,E2 -25220.982} C_VEL
LIN {X 0,Y 176.982,Z 388.195,A -85,B 0,C 180,E1 -25225.185,E2 -25225.185} C_VEL
LIN {X 0,Y 179.665,Z 393.451,A -85,B 0,C 180,E1 -25228.103,E2 -25228.103} C_VEL
LIN {X 0,Y 182.873,Z 400.229,A -85,B 0,C 180,E1 -25231.12,E2 -25231.12} C_VEL
LIN {X 0,Y 186.324,Z 408.262,A -85,B 0,C 180,E1 -25233.985,E2 -25233.985} C_VEL
LIN {X 0,Y 189.296,Z 415.81,A -85,B 0,C 180,E1 -25236.205,E2 -25236.205} C_VEL
LIN {X 0,Y 189.98,Z 417.777,A -85,B 0,C 180,E1 -25236.7,E2 -25236.7} C_VEL
LIN {X 0,Y 187.953,Z 439.382,A -85,B 0,C 180,E1 -25237.382,E2 -25237.382} C_VEL
LIN {X 0,Y 185.494,Z 453.152,A -85,B 0,C 180,E1 -25238.084,E2 -25238.084} C_VEL
LIN {X 0,Y 182.446,Z 464.65,A -85,B 0,C 180,E1 -25238.932,E2 -25238.932} C_VEL
LIN {X 0,Y 178.148,Z 476.763,A -85,B 0,C 180,E1 -25240.149,E2 -25240.149} C_VEL
LIN {X 0,Y 173.07,Z 488.216,A -85,B 0,C 180,E1 -25241.739,E2 -25241.739} C_VEL
LIN {X 0,Y 167.61,Z 498.548,A -85,B 0,C 180,E1 -25243.67,E2 -25243.67} C_VEL
LIN {X 0,Y 161.805,Z 507.875,A -85,B 0,C 180,E1 -25245.974,E2 -25245.974} C_VEL
LIN {X 0,Y 155.219,Z 516.909,A -85,B 0,C 180,E1 -25248.963,E2 -25248.963} C_VEL
LIN {X 0,Y 149.164,Z 524.214,A -85,B 0,C 180,E1 -25252.227,E2 -25252.227} C_VEL
LIN {X 0,Y 143.791,Z 530.095,A -85,B 0,C 180,E1 -25255.798,E2 -25255.798} C_VEL
LIN {X 0,Y 139.113,Z 534.762,A -85,B 0,C 180,E1 -25259.653,E2 -25259.653} C_VEL
LIN {X 0,Y 134.978,Z 538.352,A -85,B 0,C 180,E1 -25263.73,E2 -25263.73} C_VEL
LIN {X 0,Y 131.62,Z 540.964,A -85,B 0,C 180,E1 -25268.05,E2 -25268.05} C_VEL
LIN {X 0,Y 129.8,Z 542.216,A -85,B 0,C 180,E1 -25271.04,E2 -25271.04} C_VEL
LIN {X 0,Y 128.498,Z 543.059,A -85,B 0,C 180,E1 -25274.127,E2 -25274.127} C_VEL
LIN {X 0,Y 126.853,Z 543.564,A -85,B 0,C 180,E1 -25280.43,E2 -25280.43} C_VEL
LIN {X 0,Y 126.545,Z 543.254,A -85,B 0,C 180,E1 -25283.62,E2 -25283.62} C_VEL
LIN {X 0,Y 126.544,Z 541.967,A -85,B 0,C 180,E1 -25288.566,E2 -25288.566} C_VEL
LIN {X 0,Y 126.533,Z 540.854,A -85,B 0,C 180,E1 -25291.229,E2 -25291.229} C_VEL
LIN {X 0,Y 126.561,Z 537.816,A -85,B 0,C 180,E1 -25296.374,E2 -25296.374} C_VEL
LIN {X 0,Y 127.098,Z 533.874,A -85,B 0,C 180,E1 -25301.157,E2 -25301.157} C_VEL
LIN {X 0,Y 128.475,Z 527.762,A -85,B 0,C 180,E1 -25306.687,E2 -25306.687} C_VEL
LIN {X 0,Y 130.697,Z 521.06,A -85,B 0,C 180,E1 -25311.28,E2 -25311.28} C_VEL
LIN {X 0,Y 131.289,Z 519.147,A -85,B 0,C 180,E1 -25312.414,E2 -25312.414} C_VEL
LIN {X 0,Y 131.371,Z 516.763,A -85,B 0,C 180,E1 -25313.811,E2 -25313.811} C_VEL
LIN {X 0,Y 128.758,Z 508.693,A -85,B 0,C 180,E1 -25318.448,E2 -25318.448} C_VEL
LIN {X 0,Y 129.2,Z 505.909,A -85,B 0,C 180,E1 -25319.699,E2 -25319.699} C_VEL
LIN {X 0,Y 132.705,Z 495.7,A -85,B 0,C 180,E1 -25323.327,E2 -25323.327} C_VEL
LIN {X 0,Y 135.927,Z 485.727,A -85,B 0,C 180,E1 -25326.022,E2 -25326.022} C_VEL
LIN {X 0,Y 139.048,Z 474.883,A -85,B 0,C 180,E1 -25328.251,E2 -25328.251} C_VEL
LIN {X 0,Y 141.741,Z 462.879,A -85,B 0,C 180,E1 -25330.131,E2 -25330.131} C_VEL
LIN {X 0,Y 144.105,Z 449.969,A -85,B 0,C 180,E1 -25331.523,E2 -25331.523} C_VEL
LIN {X 0,Y 145.568,Z 437.238,A -85,B 0,C 180,E1 -25332.405,E2 -25332.405} C_VEL
LIN {X 0,Y 148.013,Z 396.625,A -85,B 0,C 180,E1 -25334.2,E2 -25334.2} C_VEL
LIN {X 0,Y 147.103,Z 383.995,A -85,B 0,C 180,E1 -25335.259,E2 -25335.259} C_VEL
LIN {X 0,Y 142.645,Z 371.045,A -85,B 0,C 180,E1 -25337.574,E2 -25337.574} C_VEL
LIN {X 0,Y 138.214,Z 360.761,A -85,B 0,C 180,E1 -25339.93,E2 -25339.93} C_VEL
LIN {X 0,Y 135.663,Z 355.845,A -85,B 0,C 180,E1 -25341.328,E2 -25341.328} C_VEL
LIN {X 0,Y 130.659,Z 348.309,A -85,B 0,C 180,E1 -25344.158,E2 -25344.158} C_VEL
LIN {X 0,Y 128.162,Z 344.699,A -85,B 0,C 180,E1 -25345.693,E2 -25345.693} C_VEL
LIN {X 0,Y 125.932,Z 341.535,A -85,B 0,C 180,E1 -25347.154,E2 -25347.154} C_VEL
LIN {X 0,Y 125.338,Z 340.515,A -85,B 0,C 180,E1 -25347.575,E2 -25347.575} C_VEL
LIN {X 0,Y 123.089,Z 338.414,A -85,B 0,C 180,E1 -25349.078,E2 -25349.078} C_VEL
LIN {X 0,Y 122.097,Z 336.111,A -85,B 0,C 180,E1 -25349.91,E2 -25349.91} C_VEL
LIN {X 0,Y 121.957,Z 335.29,A -85,B 0,C 180,E1 -25350.128,E2 -25350.128} C_VEL
LIN {X 0,Y 122.018,Z 335.285,A -85,B 0,C 180,E1 -25357.148,E2 -25357.148} C_VEL
LIN {X 0,Y 122.105,Z 335.24,A -85,B 0,C 180,E1 -25363.275,E2 -25363.275} C_VEL
LIN {X 0,Y 122.357,Z 335.242,A -85,B 0,C 180,E1 -25367.526,E2 -25367.526} C_VEL
LIN {X 0,Y 122.441,Z 335.222,A -85,B 0,C 180,E1 -25370.085,E2 -25370.085} C_VEL
LIN {X 0,Y 122.598,Z 335.188,A -85,B 0,C 180,E1 -25376.714,E2 -25376.714} C_VEL
LIN {X 0,Y 123.034,Z 335.157,A -85,B 0,C 180,E1 -25380,E2 -25380} C_VEL
LIN {X 0,Y 122.395,Z 335.193,A -85,B 0,C 180,E1 -25386.804,E2 -25386.804} C_VEL
LIN {X 0,Y 122.306,Z 335.25,A -85,B 0,C 180,E1 -25392.363,E2 -25392.363} C_VEL
LIN {X 0,Y 122.099,Z 335.268,A -85,B 0,C 180,E1 -25396.726,E2 -25396.726} C_VEL
LIN {X 0,Y 122.017,Z 335.277,A -85,B 0,C 180,E1 -25402.851,E2 -25402.851} C_VEL
LIN {X 0,Y 121.951,Z 335.283,A -85,B 0,C 180,E1 -25407.454,E2 -25407.454} C_VEL
LIN {X 0,Y 121.899,Z 335.298,A -85,B 0,C 180,E1 -25411.258,E2 -25411.258} C_VEL
LIN {X 0,Y 121.877,Z 335.3,A -85,B 0,C 180,E1 -25416.172,E2 -25416.172} C_VEL
LIN {X 0,Y 121.858,Z 335.304,A -85,B 0,C 180,E1 -25421.435,E2 -25421.435} C_VEL
LIN {X 0,Y 121.843,Z 335.351,A -85,B 0,C 180,E1 -25424.462,E2 -25424.462} C_VEL
LIN {X 0,Y 122.822,Z 338.087,A -85,B 0,C 180,E1 -25425.337,E2 -25425.337} C_VEL
LIN {X 0,Y 124.869,Z 340.267,A -85,B 0,C 180,E1 -25426.746,E2 -25426.746} C_VEL
LIN {X 0,Y 125.535,Z 340.969,A -85,B 0,C 180,E1 -25427.184,E2 -25427.184} C_VEL
LIN {X 0,Y 127.683,Z 344.304,A -85,B 0,C 180,E1 -25428.635,E2 -25428.635} C_VEL
LIN {X 0,Y 129.041,Z 345.942,A -85,B 0,C 180,E1 -25429.467,E2 -25429.467} C_VEL
LIN {X 0,Y 135.19,Z 355.057,A -85,B 0,C 180,E1 -25433.013,E2 -25433.013} C_VEL
LIN {X 0,Y 139.92,Z 363.106,A -85,B 0,C 180,E1 -25435.495,E2 -25435.495} C_VEL
LIN {X 0,Y 144.773,Z 372.463,A -85,B 0,C 180,E1 -25437.854,E2 -25437.854} C_VEL
LIN {X 0,Y 148.852,Z 381.558,A -85,B 0,C 180,E1 -25439.736,E2 -25439.736} C_VEL
LIN {X 0,Y 148.194,Z 394.033,A -85,B 0,C 180,E1 -25440.299,E2 -25440.299} C_VEL
LIN {X 0,Y 145.587,Z 431.472,A -85,B 0,C 180,E1 -25441.918,E2 -25441.918} C_VEL
LIN {X 0,Y 143.889,Z 445.323,A -85,B 0,C 180,E1 -25443.062,E2 -25443.062} C_VEL
LIN {X 0,Y 141.6,Z 457.074,A -85,B 0,C 180,E1 -25444.46,E2 -25444.46} C_VEL
LIN {X 0,Y 138.885,Z 469.018,A -85,B 0,C 180,E1 -25446.518,E2 -25446.518} C_VEL
LIN {X 0,Y 135.824,Z 480.562,A -85,B 0,C 180,E1 -25449.204,E2 -25449.204} C_VEL
LIN {X 0,Y 132.441,Z 490.799,A -85,B 0,C 180,E1 -25452.237,E2 -25452.237} C_VEL
LIN {X 0,Y 129.099,Z 500.09,A -85,B 0,C 180,E1 -25455.822,E2 -25455.822} C_VEL
LIN {X 0,Y 125.753,Z 509.107,A -85,B 0,C 180,E1 -25460.351,E2 -25460.351} C_VEL
LIN {X 0,Y 123.105,Z 516.371,A -85,B 0,C 180,E1 -25465.09,E2 -25465.09} C_VEL
LIN {X 0,Y 121.181,Z 522.162,A -85,B 0,C 180,E1 -25470.002,E2 -25470.002} C_VEL
LIN {X 0,Y 119.935,Z 526.7,A -85,B 0,C 180,E1 -25475.01,E2 -25475.01} C_VEL
LIN {X 0,Y 119.13,Z 530.219,A -85,B 0,C 180,E1 -25480.196,E2 -25480.196} C_VEL
LIN {X 0,Y 118.986,Z 531.959,A -85,B 0,C 180,E1 -25483.668,E2 -25483.668} C_VEL
LIN {X 0,Y 119.51,Z 534.007,A -85,B 0,C 180,E1 -25489.794,E2 -25489.794} C_VEL
LIN {X 0,Y 120.464,Z 534.668,A -85,B 0,C 180,E1 -25494.106,E2 -25494.106} C_VEL
LIN {X 0,Y 121.639,Z 534.724,A -85,B 0,C 180,E1 -25497.533,E2 -25497.533} C_VEL
LIN {X 0,Y 123.353,Z 534.32,A -85,B 0,C 180,E1 -25501.282,E2 -25501.282} C_VEL
LIN {X 0,Y 127.301,Z 532.346,A -85,B 0,C 180,E1 -25507.396,E2 -25507.396} C_VEL
LIN {X 0,Y 130.466,Z 530.324,A -85,B 0,C 180,E1 -25511.048,E2 -25511.048} C_VEL
LIN {X 0,Y 134.456,Z 527.272,A -85,B 0,C 180,E1 -25514.884,E2 -25514.884} C_VEL
LIN {X 0,Y 140.262,Z 522.202,A -85,B 0,C 180,E1 -25519.354,E2 -25519.354} C_VEL
LIN {X 0,Y 146.642,Z 515.65,A -85,B 0,C 180,E1 -25523.397,E2 -25523.397} C_VEL
LIN {X 0,Y 153.166,Z 508.072,A -85,B 0,C 180,E1 -25526.748,E2 -25526.748} C_VEL
LIN {X 0,Y 159.157,Z 499.966,A -85,B 0,C 180,E1 -25529.44,E2 -25529.44} C_VEL
LIN {X 0,Y 165.031,Z 490.737,A -85,B 0,C 180,E1 -25531.738,E2 -25531.738} C_VEL
LIN {X 0,Y 170.34,Z 480.718,A -85,B 0,C 180,E1 -25533.684,E2 -25533.684} C_VEL
LIN {X 0,Y 175.06,Z 469.994,A -85,B 0,C 180,E1 -25535.275,E2 -25535.275} C_VEL
LIN {X 0,Y 179.072,Z 458.749,A -85,B 0,C 180,E1 -25536.523,E2 -25536.523} C_VEL
LIN {X 0,Y 182.481,Z 445.851,A -85,B 0,C 180,E1 -25537.569,E2 -25537.569} C_VEL
LIN {X 0,Y 184.703,Z 433.592,A -85,B 0,C 180,E1 -25538.24,E2 -25538.24} C_VEL
LIN {X 0,Y 186.659,Z 414.11,A -85,B 0,C 180,E1 -25538.888,E2 -25538.888} C_VEL
LIN {X 0,Y 182.912,Z 406.599,A -85,B 0,C 180,E1 -25541.809,E2 -25541.809} C_VEL
LIN {X 0,Y 178.883,Z 399.377,A -85,B 0,C 180,E1 -25545.422,E2 -25545.422} C_VEL
LIN {X 0,Y 176.291,Z 395.147,A -85,B 0,C 180,E1 -25548.138,E2 -25548.138} C_VEL
LIN {X 0,Y 174.467,Z 392.135,A -85,B 0,C 180,E1 -25550.358,E2 -25550.358} C_VEL
LIN {X 0,Y 172.089,Z 388.084,A -85,B 0,C 180,E1 -25553.956,E2 -25553.956} C_VEL
LIN {X 0,Y 170.082,Z 384.993,A -85,B 0,C 180,E1 -25558.119,E2 -25558.119} C_VEL
LIN {X 0,Y 169.668,Z 383.736,A -85,B 0,C 180,E1 -25559.464,E2 -25559.464} C_VEL
LIN {X 0,Y 168.418,Z 383.104,A -85,B 0,C 180,E1 -25564.787,E2 -25564.787} C_VEL
LIN {X 0,Y 168.525,Z 383.184,A -85,B 0,C 180,E1 -25569.602,E2 -25569.602} C_VEL
LIN {X 0,Y 169.596,Z 384.168,A -85,B 0,C 180,E1 -25574.028,E2 -25574.028} C_VEL
LIN {X 0,Y 171.175,Z 387.503,A -85,B 0,C 180,E1 -25578.066,E2 -25578.066} C_VEL
LIN {X 0,Y 172.528,Z 389.118,A -85,B 0,C 180,E1 -25580.385,E2 -25580.385} C_VEL
LIN {X 0,Y 175.22,Z 394.474,A -85,B 0,C 180,E1 -25584.275,E2 -25584.275} C_VEL
LIN {X 0,Y 177.592,Z 399.404,A -85,B 0,C 180,E1 -25587.056,E2 -25587.056} C_VEL
LIN {X 0,Y 180.579,Z 406.09,A -85,B 0,C 180,E1 -25590.082,E2 -25590.082} C_VEL
LIN {X 0,Y 183.715,Z 413.831,A -85,B 0,C 180,E1 -25592.884,E2 -25592.884} C_VEL
LIN {X 0,Y 186.179,Z 420.527,A -85,B 0,C 180,E1 -25594.897,E2 -25594.897} C_VEL
LIN {X 0,Y 184.231,Z 439.955,A -85,B 0,C 180,E1 -25595.524,E2 -25595.524} C_VEL
LIN {X 0,Y 181.787,Z 453.069,A -85,B 0,C 180,E1 -25596.195,E2 -25596.195} C_VEL
LIN {X 0,Y 178.728,Z 464.23,A -85,B 0,C 180,E1 -25597,E2 -25597} C_VEL
LIN {X 0,Y 174.359,Z 476.274,A -85,B 0,C 180,E1 -25598.185,E2 -25598.185} C_VEL
LIN {X 0,Y 169.11,Z 487.768,A -85,B 0,C 180,E1 -25599.749,E2 -25599.749} C_VEL
LIN {X 0,Y 164.025,Z 497.073,A -85,B 0,C 180,E1 -25601.423,E2 -25601.423} C_VEL
LIN {X 0,Y 157.953,Z 506.63,A -85,B 0,C 180,E1 -25603.693,E2 -25603.693} C_VEL
LIN {X 0,Y 152.178,Z 514.486,A -85,B 0,C 180,E1 -25606.15,E2 -25606.15} C_VEL
LIN {X 0,Y 145.679,Z 522.196,A -85,B 0,C 180,E1 -25609.36,E2 -25609.36} C_VEL
